    PROC  WELD_A_SQUARE_ANCHOR()
        !!!NOW HAS THE WOBJ WRINKLE REMOVED 02-05-18!!!!!!!
        !!!!!THIS PROGRAM IS now revised Square_Anchor TO GET SEARCHED IN POSITION 02-05-18!!!!!!!
        !!!!! nozzle search version 02-05-18!!!!!!!!!!!
        !!!!!!!!!!!!!!!!REVISED 03-16-18 to add anchor_back X searches!!!!!
        ActUnit STN1;
		AccSet 40, 40;
        MoveJ pjthomeSTA1zero, vCellSpeed, fine, tWeldGun\WObj:=wobj0;
        MoveJ Offs(SP_AGBY_S,0,-300,50), v400, z5, tWeldGun\WObj:=wobjHanchor_BACK;
		MoveL Offs(SP_AGBY_S,0,-100,50), v300, z5, tWeldGun\WObj:=wobjHanchor_BACK;
        MoveL SP_AGBY_S, v200, z5, tWeldGun\WObj:=wobjHanchor_BACK;
		Search_1D SR_AGB_Y\SearchStop:=AG_BY, SP_AGBY_S, SP_AGBY_E, v50, tWeldGun\WObj:=wobjHanchor_BACK\SchSpeed:=10;
  		MoveL AG_BY, v50, fine, tWeldGun\WObj:=wobjHanchor_BACK;
  		WaitTime\InPos, 1;
  		AG_BY_DEFLECTION := CRobT(\Tool:=tWeldGun\WObj:=obSTN1);
  		WaitTime\InPos, 1;
		AG_BY_DEFLECTION.trans.y := AG_BY_DEFLECTION.trans.y + NOZZLE_RADIUS;
        WaitTime\InPos, 0.2;
        TPWrite "SR_AGB_Y DEFLECTION:="\Pos:=SR_AGB_Y.trans;
		MoveL SP_AGBY_S, v300, z5, tWeldGun\WObj:=wobjHanchor_BACK;
        MoveL SP_AHBY_S, v300, z5, tWeldGun\WObj:=wobjHanchor_BACK;
		Search_1D SR_AHB_Y\SearchStop:=AH_BY, SP_AHBY_S, SP_AHBY_E, v50, tWeldGun\WObj:=wobjHanchor_BACK\SchSpeed:=10;
  		MoveL AH_BY, v50, fine, tWeldGun\WObj:=wobjHanchor_BACK;
  		WaitTime\InPos, 1;
		AH_BY_DEFLECTION := CRobT(\Tool:=tWeldGun\WObj:=obSTN1);
  		WaitTime\InPos, 1;
		AH_BY_DEFLECTION.trans.y := AH_BY_DEFLECTION.trans.y + NOZZLE_RADIUS;
        WaitTime\InPos, 0.2;
		TPWrite "SR_AHB_Y DEFLECTION:="\Pos:=SR_AHB_Y.trans;
		MoveL SP_AHBY_S, v200, z5, tWeldGun\WObj:=wobjHanchor_BACK;
	    MoveJ Offs(SP_AHBY_S,0,-275,75), v500, z5, tWeldGun\WObj:=wobjHanchor_BACK;
	    MoveJ Offs(SP_AHBY_S,0,-425,125), v500, z5, tWeldGun\WObj:=wobjHanchor_BACK;
	    MoveJ Offs(SP_AHBY_S,0,-625,125), v500, z5, tWeldGun\WObj:=wobjHanchor_BACK;
		MoveJ Offs(SP_GX_S,0,-400,50), v500, z5, tWeldGun\WObj:=wobjHanchor_BACK;
		MoveJ Offs(SP_GX_S,0,-200,50), v500, z5, tWeldGun\WObj:=wobjHanchor_BACK;
		MoveL Offs(SP_GX_S,0,-200,50), v500, z5, tWeldGun\WObj:=wobjHanchor_BACK;
		MoveL Offs(SP_GX_S,0,-50,50), v500, z5, tWeldGun\WObj:=wobjHanchor_BACK;
        MoveL SP_GX_S, v200, z1, tWeldGun\WObj:=wobjHanchor;
		Search_1D SR_AG_X\SearchStop:=AG_X, SP_GX_S, SP_GX_E, v50, tWeldGun\WObj:=wobjHanchor\SchSpeed:=10;
        TPWrite "SR_AG_X :="\Pos:=SR_AG_X.trans;
		MoveL SP_GX_S, v200, z1, tWeldGun\WObj:=wobjHanchor;
        MoveL SP_AGBZ_S, v200, z1, tWeldGun\WObj:=wobjHanchor_BACK;
	    Search_1D SR_AGB_Z\SearchStop:=AG_BZ, SP_AGBZ_S, SP_AGBZ_E, v50, tWeldGun\WObj:=wobjHanchor_BACK\SchSpeed:=10;
     	MoveL AG_BZ, v50, fine, tWeldGun\WObj:=wobjHanchor_BACK;
  		WaitTime\InPos, 1;
		AG_BZ_DEFLECTION := CRobT(\Tool:=tWeldGun\WObj:=obSTN1);
        WaitTime\InPos, .1;
        TPWrite "SR_AGB_Z DEFLECTION:="\Pos:=SR_AGB_Z.trans;
        MoveL SP_AGBZ_S, v200, z1, tWeldGun\WObj:=wobjHanchor_BACK;
        MoveL Offs(SP_AGBZ_S,0,-325,50), v200, z1, tWeldGun\WObj:=wobjHanchor_BACK;
        MoveJ Offs(SP_AHBZ_S,0,-325,50), v200, z1, tWeldGun\WObj:=wobjHanchor_BACK;
        MoveL SP_AHBZ_S, v200, z1, tWeldGun\WObj:=wobjHanchor_BACK;
	    Search_1D SR_AHB_Z\SearchStop:=AH_BZ, SP_AHBZ_S, SP_AHBZ_E, v50, tWeldGun\WObj:=wobjHanchor_BACK\SchSpeed:=10;
     	MoveL AH_BZ, v50, fine, tWeldGun\WObj:=wobjHanchor_BACK;
  		WaitTime\InPos, 1;
		AH_BZ_DEFLECTION := CRobT(\Tool:=tWeldGun\WObj:=obSTN1);
        WaitTime\InPos, .1;
        TPWrite "SR_AHB_Z DEFLECTION:="\Pos:=SR_AHB_Z.trans;
        MoveL SP_AHBZ_S, v200, z1, tWeldGun\WObj:=wobjHanchor_BACK;
        MoveL SP_HX_S, v200, z1, tWeldGun\WObj:=wobjHanchor;
		Search_1D SR_AH_X\SearchStop:=AH_X, SP_HX_S, SP_HX_E, v50, tWeldGun\WObj:=wobjHanchor\SchSpeed:=10;
        TPWrite "SR_AH_X :="\Pos:=SR_AH_X.trans;
		MoveL SP_HX_S, v200, z1, tWeldGun\WObj:=wobjHanchor;
		MoveL Offs(SP_AHBZ_S,0,-125,50), v200, z5, tWeldGun\WObj:=wobjHanchor_BACK;
		MoveL Offs(SP_AHBZ_S,0,-500,100), v200, z5, tWeldGun\WObj:=wobjHanchor_BACK;
        RESET_ANCHOR_BACK_WOBJ;
        SET_ANCHOR_X AH_X ;
        SET_ANCHOR_X AG_X ;
        TPWrite "NOW WORKING ON WELD 'AH_BACK'";
		MoveJ Offs(AH201,-150,-250,-10), vExtMax, z1, tWeldGun\WObj:=wobjHanchor_BACK_H;
		MoveL RelTool(AH200,0,0,-20), v200, z1, tWeldGun\WObj:=wobjHanchor_BACK_H;
		ArcLStart AH200, v100, smHCYLANCH, wdHCYLANCH\Weave:=wvHCYLANCH, fine, tWeldGun\WObj:=wobjHanchor_BACK_H\Track:=trHCYLANCHhiteonly;
		ArcL AH201, v100, smHCYLANCH, wdHCYLANCH\Weave:=wvHCYLANCH, z10, tWeldGun\WObj:=wobjHanchor_BACK_H\Track:=trHCYLANCHhiteonly;
		ArcLEnd AH202, v100, smHCYLANCH, wdHCYLANCH\Weave:=wvHCYLANCH, z10, tWeldGun\WObj:=wobjHanchor_BACK_H\Track:=trHCYLANCHhiteonly;
		MoveL RelTool(AH202,0,0,-100), v200, z1, tWeldGun\WObj:=wobjHanchor_BACK;
		MoveJ Offs(AH202,-50,-150,0), vExtMax, z1, tWeldGun\WObj:=wobjHanchor_BACK;
	    TPWrite "NOW WORKING ON WELD 'AG_BACK'";
		MoveL Offs(AG201,50,-150,0), vExtMax, z1, tWeldGun\WObj:=wobjHanchor_BACK;
		MoveL RelTool(AG200,0,0,-20), v200, z1, tWeldGun\WObj:=wobjHanchor_BACK;
		ArcLStart AG200, v100, smHCYLANCH, wdHCYLANCH\Weave:=wvHCYLANCH, fine, tWeldGun\WObj:=wobjHanchor_BACK_G\Track:=trHCYLANCHhiteonly;
		ArcL AG201, v100, smHCYLANCH, wdHCYLANCH\Weave:=wvHCYLANCH, z10, tWeldGun\WObj:=wobjHanchor_BACK_G\Track:=trHCYLANCHhiteonly;
		ArcLEnd AG202, v100, smHCYLANCH, wdHCYLANCH\Weave:=wvHCYLANCH, z10, tWeldGun\WObj:=wobjHanchor_BACK_G\Track:=trHCYLANCHhiteonly;
		MoveL RelTool(AG202,0,0,-100), v200, z1, tWeldGun\WObj:=wobjHanchor_BACK;
		MoveL pairanchor11, v500, z1, tWeldGun\WObj:=wobjHanchor_BACK;
		MoveJ pjthomeSTA1zero, vCellSpeed, fine, tWeldGun\WObj:=wobj0;
		!MoveL Offs(AG202,300,-650,50), v200, z1, tWeldGun\WObj:=wobjHanchor_BACK;
		!CutWire;
		ActUnit STN1;
        MoveJ Offs(SP_AGFY_S,0,800,200), v1000, z5, tWeldGun\WObj:=wobjHanchor_FRONT;
        MoveJ Offs(SP_AGFY_S,0,150,100), v400, z5, tWeldGun\WObj:=wobjHanchor_FRONT;
        MoveL SP_AGFY_S, v200, z1, tWeldGun\WObj:=wobjHanchor_FRONT;
		Search_1D SR_AGF_Y1\SearchStop:=AG_FY, SP_AGFY_S, SP_AGFY_E, v50, tWeldGun\WObj:=wobjHanchor_FRONT\SchSpeed:=10;
        TPWrite "SR_AGF_Y1 DEFLECTION:="\Pos:=SR_AGF_Y1.trans;
		Search_1D SR_AGF_Y2\SearchStop:=AG_FY, SP_AGFY_S, SP_AGFY_E, v50, tWeldGun\WObj:=wobjHanchor_FRONT\SchSpeed:=10;
        TPWrite "SR_AGF_Y2 DEFLECTION:="\Pos:=SR_AGF_Y2.trans;
        MoveL AG_FY, v50, fine, tWeldGun\WObj:=wobjHanchor_FRONT;
  		WaitTime\InPos, 1;
		AG_FY_DEFLECTION := CRobT(\Tool:=tWeldGun\WObj:=obSTN1);
        WaitTime\InPos, 1;
        AG_FY_DEFLECTION.trans.y := AG_FY_DEFLECTION.trans.y - NOZZLE_RADIUS;
        WaitTime\InPos, 0.2;
		MoveL SP_AGFY_S, v300, z1, tWeldGun\WObj:=wobjHanchor_FRONT;
        MoveL SP_AHFY_S, v300, z1, tWeldGun\WObj:=wobjHanchor_FRONT;
		Search_1D SR_AHF_Y1\SearchStop:=AH_FY, SP_AHFY_S, SP_AHFY_E, v50, tWeldGun\WObj:=wobjHanchor_FRONT\SchSpeed:=10;
        TPWrite "SR_AHF_Y1 DEFLECTION:="\Pos:=SR_AHF_Y1.trans;
		Search_1D SR_AHF_Y2\SearchStop:=AH_FY, SP_AHFY_S, SP_AHFY_E, v50, tWeldGun\WObj:=wobjHanchor_FRONT\SchSpeed:=10;
  		TPWrite "SR_AHF_Y2 DEFLECTION:="\Pos:=SR_AHF_Y2.trans;
        MoveL AH_FY, v50, fine, tWeldGun\WObj:=wobjHanchor_FRONT;
  		WaitTime\InPos, 1;
		AH_FY_DEFLECTION := CRobT(\Tool:=tWeldGun\WObj:=obSTN1);
        WaitTime\InPos, 1;
        AH_FY_DEFLECTION.trans.y := AH_FY_DEFLECTION.trans.y - NOZZLE_RADIUS;
        WaitTime\InPos, 0.2;
	    ! POSSIBLY NEED TO ADD A "Y" DISPLACEMENT TO KEEP THE "Z" SEARCH ON THE NOZZLE
        SR_AHF_Y2.TRANS.Y := SR_AHF_Y1.TRANS.Y;
		PDispSet SR_AHF_Y2;
		MoveL Offs(SP_AHFY_S,0,50,0), v300, z1, tWeldGun\WObj:=wobjHanchor_FRONT;
		MoveL Offs(SP_AHFY_S,0,250,100), v300, z1, tWeldGun\WObj:=wobjHanchor_FRONT;
        MoveJ Offs(SP_AHFZ_S,0,400,50), v300, z1, tWeldGun\WObj:=wobjHanchor_FRONT;
        MoveJ Offs(SP_AHFZ_S,0,100,50), v300, z1, tWeldGun\WObj:=wobjHanchor_FRONT;
		MoveL SP_AHFZ_S, v200, z1, tWeldGun\WObj:=wobjHanchor_FRONT;
        Search_1D SR_AHF_Z\SearchStop:=AH_FZ, SP_AHFZ_S, SP_AHFZ_E, v50, tWeldGun\WObj:=wobjHanchor_FRONT\SchSpeed:=10;
  		MoveL AH_FZ, v50, fine, tWeldGun\WObj:=wobjHanchor_FRONT;
        WaitTime\InPos, 1;
        AH_FZ_DEFLECTION := CRobT(\Tool:=tWeldGun\WObj:=obSTN1);
        WaitTime\InPos, 1;
        TPWrite "SR_AGF_Z DEFLECTION:="\Pos:=SR_AGF_Z.trans;
		MoveL SP_AHFZ_S, v200, z1, tWeldGun\WObj:=wobjHanchor_FRONT;
        ! ADDED X SEARCH HERE
		MoveJ SP_AHFX_S, v200, z1, tWeldGun\WObj:=wobjHanchor_FRONT;
        Search_1D SR_AHF_X\SearchStop:=AH_X, SP_AHFX_S, SP_AHFX_E, v50, tWeldGun\WObj:=wobjHanchor_FRONT\SchSpeed:=10;
		MoveL SP_AHFZ_S, v200, z1, tWeldGun\WObj:=wobjHanchor_FRONT;
        ! POSSIBLY NEED TO ADD A "Y" DISPLACEMENT TO KEEP THE "Z" SEARCH ON THE NOZZLE
        SR_AGF_Y2.TRANS.Y := SR_AGF_Y1.TRANS.Y;
		PDispSet SR_AGF_Y2;
        MoveJ SP_AGFZ_S, v200, z1, tWeldGun\WObj:=wobjHanchor_FRONT;
		Search_1D SR_AGF_Z\SearchStop:=AG_FZ, SP_AGFZ_S, SP_AGFZ_E, v50, tWeldGun\WObj:=wobjHanchor_FRONT\SchSpeed:=10;
   		MoveL AG_FZ, v50, fine, tWeldGun\WObj:=wobjHanchor_FRONT;
        WaitTime\InPos, 1;
        AG_FZ_DEFLECTION := CRobT(\Tool:=tWeldGun\WObj:=obSTN1);
        WaitTime\InPos, 1;
        TPWrite "SR_AGF_Z DEFLECTION:="\Pos:=SR_AGF_Z.trans;
		MoveL SP_AGFZ_S, v200, z1, tWeldGun\WObj:=wobjHanchor_FRONT;
        ! ADDED X SEARCH HERE
 		MoveL SP_AGFX_S, v200, z1, tWeldGun\WObj:=wobjHanchor_FRONT;
        Search_1D SR_AGF_X\SearchStop:=AG_X, SP_AGFX_S, SP_AGFX_E, v50, tWeldGun\WObj:=wobjHanchor_FRONT\SchSpeed:=10;
		MoveL SP_AGFZ_S, v200, z1, tWeldGun\WObj:=wobjHanchor_FRONT;
        MoveL OFFS(SP_AGFZ_S,0,100,75), v200, z1, tWeldGun\WObj:=wobjHanchor_FRONT;
        MoveL OFFS(SP_AGFZ_S,0,600,75), v400, z1, tWeldGun\WObj:=wobjHanchor_FRONT;
        FRONT_ANCHOR_ROTATION_DEFLECTION  wobjHanchor_FRONT_H, AH_FY_DEFLECTION, AH_FY, AH_FZ_DEFLECTION, AH_FZ;
        FRONT_ANCHOR_ROTATION_DEFLECTION  wobjHanchor_FRONT_G, AG_FY_DEFLECTION, AG_FY, AG_FZ_DEFLECTION, AG_FZ;
        FRONT_ANCHOR_TRANS_DEFLECTION wobjHanchor_FRONT_G, AG_FY_DEFLECTION, AG_FZ_DEFLECTION, AG_FY, AG_FZ  ;
        FRONT_ANCHOR_TRANS_DEFLECTION wobjHanchor_FRONT_H, AH_FY_DEFLECTION, AH_FZ_DEFLECTION, AH_FY, AH_FZ  ;
        SET_ANCHOR_X AG_X;
        SET_ANCHOR_X AH_X;
        MoveJ Offs(AG206,150,300,50), v400, z1, tWeldGun\WObj:=wobjHanchor_FRONT_G;
		MoveL RelTool(AG206,0,0,-30), v200, z1, tWeldGun\WObj:=wobjHanchor_FRONT_G;
        ArcLStart AG206, v100, smHCYLANCH, wdHCYLANCH\Weave:=wvHCYLANCH, fine, tWeldGun\WObj:=wobjHanchor_FRONT_G\Track:=trHCYLANCHhiteonly;
		ArcL AG207, v100, smHCYLANCH, wdHCYLANCH\Weave:=wvHCYLANCH, z10, tWeldGun\WObj:=wobjHanchor_FRONT_G\Track:=trHCYLANCHhiteonly;
		ArcLEnd AG208, v100, smHCYLANCH, wdHCYLANCH\Weave:=wvHCYLANCH, z10, tWeldGun\WObj:=wobjHanchor_FRONT_G\Track:=trHCYLANCHhiteonly;
		MoveL RelTool(AG208,0,0,-10), v200, z1, tWeldGun\WObj:=wobjHanchor_FRONT_G;
		MoveL RelTool(AG206,0,0,-150), vExtMax, z1, tWeldGun\WObj:=wobjHanchor_FRONT_G;
		MoveL Offs(AG206,150,250,50), vExtMax, z1, tWeldGun\WObj:=wobjHanchor_FRONT_G;
		MoveJ Offs(AG220,150,350,50), vExtMax, z1, tWeldGun\WObj:=wobjHanchor_FRONT_G;
		MoveJ Offs(AG220,50,350,50), vExtMax, z1, tWeldGun\WObj:=wobjHanchor_FRONT_G;
   		MoveJ Offs(AG220,50,50,50), vExtMax, z1, tWeldGun\WObj:=wobjHanchor_FRONT_G;
    	MoveL RelTool(AG220,0,0,-15), vExtMax, fine, tWeldGun\WObj:=wobjHanchor_FRONT_G;
		ArcLStart AG220, v100, smHCYLANCH, wdHCYLANCH\Weave:=wv0, fine, tWeldGun\WObj:=wobjHanchor_FRONT_G\Track:=trHCYLANCHhiteonly;
		ArcL AG219, v100, smHCYLANCH, wdHCYLANCH\Weave:=wv0, z10, tWeldGun\WObj:=wobjHanchor_FRONT_G\Track:=trHCYLANCHhiteonly;
		ArcLEnd AG218, v100, smHCYLANCH, wdHCYLANCH\Weave:=wv0, z10, tWeldGun\WObj:=wobjHanchor_FRONT_G\Track:=trHCYLANCHhiteonly;
		MoveL RelTool(AG218,0,-5,-15), vExtMax, fine, tWeldGun\WObj:=wobjHanchor_FRONT_G;
		MoveL RelTool(AG219,0,-5,-15), vExtMax, fine, tWeldGun\WObj:=wobjHanchor_FRONT_G;
		MoveL RelTool(AG220,0,-10,-15), vExtMax, fine, tWeldGun\WObj:=wobjHanchor_FRONT_G;
  		MoveJ Offs(AG220,50,75,50), vExtMax, z1, tWeldGun\WObj:=wobjHanchor_FRONT_G;
  		MoveJ Offs(AG220,150,350,50), vExtMax, z1, tWeldGun\WObj:=wobjHanchor_FRONT_G;
  		IF bAnchor_Lite = TRUE THEN
  			GOTO Short_Cut;
  		ENDIF
        MoveJ Offs(AG203,75,350,-25), vExtMax, z1, tWeldGun\WObj:=wobjHanchor_FRONT_G;
		MoveL Offs(AG203,25,25,-25), vExtMax, z1, tWeldGun\WObj:=wobjHanchor_FRONT_G;
		MoveL RelTool(AG203,0,0,-15), vExtMax, fine, tWeldGun\WObj:=wobjHanchor_FRONT_G;
		ArcLStart AG203, v100, smHCYLANCH, wdHCYLANCH\Weave:=wvHCYLANCH, z0, tWeldGun\WObj:=wobjHanchor_FRONT_G\Track:=trHCYLANCHhiteonly;
		ArcL AG204, v100, smHCYLANCH, wdHCYLANCH\Weave:=wvHCYLANCH, z10, tWeldGun\WObj:=wobjHanchor_FRONT_G\Track:=trHCYLANCHhiteonly;
		ArcLEnd AG205, v100, smHCYLANCH, wdHCYLANCH\Weave:=wvHCYLANCH, fine, tWeldGun\WObj:=wobjHanchor_FRONT_G\Track:=trHCYLANCHhiteonly;
		MoveL RelTool(AG204,10,0,-15), vExtMax, fine, tWeldGun\WObj:=wobjHanchor_FRONT_G;
		MoveL Offs(AG204,30,100,-25), vExtMax, fine, tWeldGun\WObj:=wobjHanchor_FRONT_G;
		MoveL Offs(AG204,75,200,-40), vExtMax, fine, tWeldGun\WObj:=wobjHanchor_FRONT_G;
		Short_Cut:
		MoveL Offs(AG205,850,450,100), vExtMax, fine, tWeldGun\WObj:=wobjHanchor_FRONT_G;
 		MoveJ Offs(AH206,-150,250,100), vExtMax, z1, tWeldGun\WObj:=wobjHanchor_FRONT_H;
 		MoveL RelTool(AH206,0,0,-20), v200, z1, tWeldGun\WObj:=wobjHanchor_FRONT_H;
        ArcLStart AH206, v100, smHCYLANCH, wdHCYLANCH\Weave:=wvHCYLANCH, z0, tWeldGun\WObj:=wobjHanchor_FRONT_H\Track:=trHCYLANCHhiteonly;
		ArcL AH207, v100, smHCYLANCH, wdHCYLANCH\Weave:=wvHCYLANCH, z10, tWeldGun\WObj:=wobjHanchor_FRONT_H\Track:=trHCYLANCHhiteonly;
		ArcLEnd AH208, v100, smHCYLANCH, wdHCYLANCH\Weave:=wvHCYLANCH, fine, tWeldGun\WObj:=wobjHanchor_FRONT_H\Track:=trHCYLANCHhiteonly;
		MoveL RelTool(AH208,0,0,-10), v200, z1, tWeldGun\WObj:=wobjHanchor_FRONT_H;
		MoveL RelTool(AH206,0,0,-150), vExtMax, z1, tWeldGun\WObj:=wobjHanchor_FRONT_H;
		MoveJ Offs(AH206,-150,250,50), vExtMax, z1, tWeldGun\WObj:=wobjHanchor_FRONT_H;
		MoveJ Offs(AH220,-150,250,50), vExtMax, z1, tWeldGun\WObj:=wobjHanchor_FRONT_H;
		MoveL RelTool(AH220,-3,3,-15), vExtMax, fine, tWeldGun\WObj:=wobjHanchor_FRONT_H;
  		ArcLStart AH220, v100, smHCYLANCH, wdHCYLANCH\Weave:=wv0, fine, tWeldGun\WObj:=wobjHanchor_FRONT_H\Track:=trHCYLANCHhiteonly;
		ArcL AH219, v100, smHCYLANCH, wdHCYLANCH\Weave:=wv0, z10, tWeldGun\WObj:=wobjHanchor_FRONT_H\Track:=trHCYLANCHhiteonly;
		ArcLEnd AH218, v100, smHCYLANCH, wdHCYLANCH\Weave:=wv0, z10, tWeldGun\WObj:=wobjHanchor_FRONT_H\Track:=trHCYLANCHhiteonly;
		PDispOff;
		MoveL RelTool(AH218,-0,3,-15), v200, fine, tWeldGun\WObj:=wobjHanchor_FRONT_H;
		MoveL RelTool(AH219,-0,3,-15), v200, fine, tWeldGun\WObj:=wobjHanchor_FRONT_H;
		MoveL RelTool(AH220,-8,0,-15), v200, fine, tWeldGun\WObj:=wobjHanchor_FRONT_H;
  		MoveJ Offs(AH220,-100,250,0), vExtMax, z1, tWeldGun\WObj:=wobjHanchor_FRONT_H;
  		MoveJ Offs(AH206,-100,250,0), vExtMax, z1, tWeldGun\WObj:=wobjHanchor_FRONT_H;
  		IF bAnchor_Lite = TRUE THEN
  			GOTO Shorter_Cut;
  		ENDIF
       	MoveL Offs(AH203,-50,350,-50), vExtMax, z1, tWeldGun\WObj:=wobjHanchor_FRONT_H;
		MoveL Offs(AH203,-25,25,-25), vExtMax, z1, tWeldGun\WObj:=wobjHanchor_FRONT_H;
		MoveL RelTool(AH203,8,0,-15), v200, z1, tWeldGun\WObj:=wobjHanchor_FRONT_H;
		ArcLStart AH203, v100, smHCYLANCH, wdHCYLANCH\Weave:=wvHCYLANCH, fine, tWeldGun\WObj:=wobjHanchor_FRONT_H\Track:=trHCYLANCHhiteonly;
		ArcL AH204, v100, smHCYLANCH, wdHCYLANCH\Weave:=wvHCYLANCH, z10, tWeldGun\WObj:=wobjHanchor_FRONT_H\Track:=trHCYLANCHhiteonly;
		ArcLEnd AH205, v100, smHCYLANCH, wdHCYLANCH\Weave:=wvHCYLANCH, fine, tWeldGun\WObj:=wobjHanchor_FRONT_H\Track:=trHCYLANCHhiteonly;
		MoveL RelTool(AH204,8,0,-15), v200, z1, tWeldGun\WObj:=wobjHanchor_FRONT_H;
		MoveL RelTool(AH203,8,0,-15), v200, z1, tWeldGun\WObj:=wobjHanchor_FRONT_H;
		MoveL Offs(AH203,-50,50,-25), vExtMax, z1, tWeldGun\WObj:=wobjHanchor_FRONT_H;
		MoveL Offs(AH203,-100,150,-25), vExtMax, z1, tWeldGun\WObj:=wobjHanchor_FRONT_H;
		MoveL Offs(AH203,-250,250,-25), vExtMax, fine, tWeldGun\WObj:=wobjHanchor_FRONT_H;
		Shorter_Cut:
        MoveL Offs(AH208,-350,550,20), vExtMax, z1, tWeldGun\WObj:=wobjHanchor_FRONT_H;
        MoveJ pjthomeSTA1zero, vCellSpeed, fine, tWeldGun\WObj:=wobj0;
        LABEL:
    ENDPROC

    PROC  WELD_A_TAPERED_SQUARE_ANCHOR()
        !THE WOBJ WRINKLE HAS BEEN REMOVED FROM THIS PROC 12-01-17!!!!!!!!!!!
        !!!!!THIS PROGRAM IS now revised Tapered_Square_Anchor TO GET SEARCHED IN POSITION 12-01-17!!!!!!!
        !!!!! nozzle search version 12-01-17!!!!!!!!!!!
        !!!!!!!!!!!!!!!!REVISED 03-16-18 to add anchor_back X searches!!!!!
        ActUnit STN1;
		AccSet 40, 40;
        MoveJ pjthomeSTA1zero, vCellSpeed, fine, tWeldGun\WObj:=wobj0;
        MoveJ Offs(SP_AGBY_S,0,-300,50), v500, z5, tWeldGun\WObj:=wobjHanchor_BACK;
		MoveL Offs(SP_AGBY_S,0,-100,50), v500, z5, tWeldGun\WObj:=wobjHanchor_BACK;
        MoveL SP_AGBY_S, v500, z5, tWeldGun\WObj:=wobjHanchor_BACK;
		Search_1D SR_AGB_Y\SearchStop:=AG_BY, SP_AGBY_S, SP_AGBY_E, v50, tWeldGun\WObj:=wobjHanchor_BACK\SchSpeed:=10;
  		MoveL AG_BY, v50, fine, tWeldGun\WObj:=wobjHanchor_BACK;
  		WaitTime\InPos, 1;
		AG_BY_DEFLECTION := CRobT(\Tool:=tWeldGun\WObj:=obSTN1);
        WaitTime\InPos, 1;
        AG_BY_DEFLECTION.trans.y := AG_BY_DEFLECTION.trans.y + NOZZLE_RADIUS;
        WaitTime\InPos, 0.2;
        TPWrite "SR_AGB_Y DEFLECTION:="\Pos:=SR_AGB_Y.trans;
		MoveL SP_AGBY_S, v500, z5, tWeldGun\WObj:=wobjHanchor_BACK;
        MoveL SP_AHBY_S, v500, z5, tWeldGun\WObj:=wobjHanchor_BACK;
		Search_1D SR_AHB_Y\SearchStop:=AH_BY, SP_AHBY_S, SP_AHBY_E, v50, tWeldGun\WObj:=wobjHanchor_BACK\SchSpeed:=10;
  		MoveL AH_BY, v50, fine, tWeldGun\WObj:=wobjHanchor_BACK;
  		WaitTime\InPos, 1;
		AH_BY_DEFLECTION := CRobT(\Tool:=tWeldGun\WObj:=obSTN1);
        WaitTime\InPos, 1;
        AH_BY_DEFLECTION.trans.y := AH_BY_DEFLECTION.trans.y + NOZZLE_RADIUS;
        WaitTime\InPos, 0.2;
		TPWrite "SR_AHB_Y DEFLECTION:="\Pos:=SR_AHB_Y.trans;
		MoveL SP_AHBY_S, v500, z5, tWeldGun\WObj:=wobjHanchor_BACK;
	    MoveJ Offs(SP_AHBY_S,0,-275,75), v500, z5, tWeldGun\WObj:=wobjHanchor_BACK;
	    MoveJ Offs(SP_AHBY_S,0,-575,175), v500, z5, tWeldGun\WObj:=wobjHanchor_BACK;
	    MoveJ Offs(SP_GX_S,0,-400,150), v500, z5, tWeldGun\WObj:=wobjHanchor_BACK;
		MoveJ Offs(SP_GX_S,0,-300,50), v500, z5, tWeldGun\WObj:=wobjHanchor_BACK;
		MoveL Offs(SP_GX_S,0,-200,50), v500, z5, tWeldGun\WObj:=wobjHanchor_BACK;
		MoveL Offs(SP_GX_S,0,-50,50), v500, z5, tWeldGun\WObj:=wobjHanchor_BACK;
        MoveL SP_GX_S, v500, z1, tWeldGun\WObj:=wobjHanchor;
		Search_1D SR_AG_X\SearchStop:=AG_X, SP_GX_S, SP_GX_E, v50, tWeldGun\WObj:=wobjHanchor\SchSpeed:=10;
        TPWrite "SR_AG_X :="\Pos:=SR_AG_X.trans;
		MoveL SP_GX_S, v500, z1, tWeldGun\WObj:=wobjHanchor;
        MoveL SP_AGBZ_S, v500, z1, tWeldGun\WObj:=wobjHanchor_BACK;
	    Search_1D SR_AGB_Z\SearchStop:=AG_BZ, SP_AGBZ_S, SP_AGBZ_E, v50, tWeldGun\WObj:=wobjHanchor_BACK\SchSpeed:=10;
     	MoveL AG_BZ, v50, fine, tWeldGun\WObj:=wobjHanchor_BACK;
  		WaitTime\InPos, 1;
		AG_BZ_DEFLECTION := CRobT(\Tool:=tWeldGun\WObj:=obSTN1);
        WaitTime\InPos, 1;
        TPWrite "SR_AGB_Z DEFLECTION:="\Pos:=SR_AGB_Z.trans;
        MoveL SP_AGBZ_S, v500, z1, tWeldGun\WObj:=wobjHanchor_BACK;
        MoveL Offs(SP_AGBZ_S,100,-325,50), v500, z1, tWeldGun\WObj:=wobjHanchor_BACK;
        MoveJ Offs(SP_AHBZ_S,0,-325,50), v500, z1, tWeldGun\WObj:=wobjHanchor_BACK;
        MoveL SP_AHBZ_S, v500, z1, tWeldGun\WObj:=wobjHanchor_BACK;
	    Search_1D SR_AHB_Z\SearchStop:=AH_BZ, SP_AHBZ_S, SP_AHBZ_E, v50, tWeldGun\WObj:=wobjHanchor_BACK\SchSpeed:=10;
     	MoveL AH_BZ, v50, fine, tWeldGun\WObj:=wobjHanchor_BACK;
  		WaitTime\InPos, 1;
		AH_BZ_DEFLECTION := CRobT(\Tool:=tWeldGun\WObj:=obSTN1);
        WaitTime\InPos, 1;
        TPWrite "SR_AHB_Z DEFLECTION:="\Pos:=SR_AHB_Z.trans;
        MoveL SP_AHBZ_S, v500, z1, tWeldGun\WObj:=wobjHanchor_BACK;
        MoveL SP_HX_S, v500, z1, tWeldGun\WObj:=wobjHanchor;
		Search_1D SR_AH_X\SearchStop:=AH_X, SP_HX_S, SP_HX_E, v50, tWeldGun\WObj:=wobjHanchor\SchSpeed:=10;
        TPWrite "SR_AH_X :="\Pos:=SR_AH_X.trans;
		MoveL SP_HX_S, v500, z1, tWeldGun\WObj:=wobjHanchor;
		MoveL Offs(SP_AHBZ_S,0,-125,50), v500, z5, tWeldGun\WObj:=wobjHanchor_BACK;
		MoveL Offs(SP_AHBZ_S,0,-500,100), v500, z5, tWeldGun\WObj:=wobjHanchor_BACK;
	    RESET_ANCHOR_BACK_WOBJ;
        SET_ANCHOR_X AG_X;
        SET_ANCHOR_X AH_X;
        TPWrite "NOW WORKING ON WELD 'AH_BACK'";
		MoveJ Offs(AH401,-150,-250,-10), vExtMax, z1, tWeldGun\WObj:=wobjHanchor_BACK_H;
		MoveL RelTool(AH400,0,0,-20), v500, z1, tWeldGun\WObj:=wobjHanchor_BACK_H;
		ArcLStart AH400, v100, smHCYLANCH, wdHCYLANCH\Weave:=wvHCYLANCH, fine, tWeldGun\WObj:=wobjHanchor_BACK_H\Track:=trHCYLANCHhiteonly;
		ArcL AH401, v100, smHCYLANCH, wdHCYLANCH\Weave:=wvHCYLANCH, z10, tWeldGun\WObj:=wobjHanchor_BACK_H\Track:=trHCYLANCHhiteonly;
		ArcLEnd AH402, v100, smHCYLANCH, wdHCYLANCH\Weave:=wvHCYLANCH, z10, tWeldGun\WObj:=wobjHanchor_BACK_H\Track:=trHCYLANCHhiteonly;
		MoveL RelTool(AH402,0,0,-100), v200, z1, tWeldGun\WObj:=wobjHanchor_BACK;
		MoveJ Offs(AH402,-50,-150,0), vExtMax, z1, tWeldGun\WObj:=wobjHanchor_BACK;
	    TPWrite "NOW WORKING ON WELD 'AG_BACK'";
		MoveL Offs(AG401,50,-150,0), vExtMax, z1, tWeldGun\WObj:=wobjHanchor_BACK;
		MoveL RelTool(AG400,0,0,-20), v500, z1, tWeldGun\WObj:=wobjHanchor_BACK;
		ArcLStart AG400, v100, smHCYLANCH, wdHCYLANCH\Weave:=wvHCYLANCH, fine, tWeldGun\WObj:=wobjHanchor_BACK_G\Track:=trHCYLANCHhiteonly;
		ArcL AG401, v100, smHCYLANCH, wdHCYLANCH\Weave:=wvHCYLANCH, z10, tWeldGun\WObj:=wobjHanchor_BACK_G\Track:=trHCYLANCHhiteonly;
		ArcLEnd AG402, v100, smHCYLANCH, wdHCYLANCH\Weave:=wvHCYLANCH, z10, tWeldGun\WObj:=wobjHanchor_BACK_G\Track:=trHCYLANCHhiteonly;
		MoveL RelTool(AG402,0,0,-100), v500, z1, tWeldGun\WObj:=wobjHanchor_BACK;
		MoveL RelTool(AG402,0,0,-300), v500, z1, tWeldGun\WObj:=wobjHanchor_BACK;
		!MoveL Offs(AG402,300,-650,50), v200, z1, tWeldGun\WObj:=wobjHanchor_BACK;
		MoveJ pjthomeSTA1zero, vCellSpeed, fine, tWeldGun\WObj:=wobj0;
		!CutWire;
		ActUnit STN1;
        !!!!!!!!!!!  WILLIE MAKE IT   !!!!!!!!!!!
        MoveJ Offs(SP_AGFY_S,0,800,0), v1000, z5, tWeldGun\WObj:=wobjHanchor_FRONT;
        !!!!!!!!!!!  WILLIE MAKE IT   !!!!!!!!!!!
        MoveJ Offs(SP_AGFY_S,0,150,0), v500, z5, tWeldGun\WObj:=wobjHanchor_FRONT;
        MoveL SP_AGFY_S, v500, z1, tWeldGun\WObj:=wobjHanchor_FRONT;
		Search_1D SR_AGF_Y1\SearchStop:=AG_FY, SP_AGFY_S, SP_AGFY_E, v50, tWeldGun\WObj:=wobjHanchor_FRONT\SchSpeed:=10;
        TPWrite "SR_AGF_Y1 DEFLECTION:="\Pos:=SR_AGF_Y1.trans;
		Search_1D SR_AGF_Y2\SearchStop:=AG_FY, SP_AGFY_S, SP_AGFY_E, v50, tWeldGun\WObj:=wobjHanchor_FRONT\SchSpeed:=10;
        TPWrite "SR_AGF_Y2 DEFLECTION:="\Pos:=SR_AGF_Y2.trans;
        MoveL AG_FY, v50, fine, tWeldGun\WObj:=wobjHanchor_FRONT;
  		WaitTime\InPos, 1;
		AG_FY_DEFLECTION := CRobT(\Tool:=tWeldGun\WObj:=obSTN1);
        WaitTime\InPos, 1;
        AG_FY_DEFLECTION.trans.y := AG_FY_DEFLECTION.trans.y - NOZZLE_RADIUS;
        WaitTime\InPos, 0.2;
        MoveL SP_AGFY_S, v500, z1, tWeldGun\WObj:=wobjHanchor_FRONT;
        MoveL SP_AHFY_S, v500, z1, tWeldGun\WObj:=wobjHanchor_FRONT;
		Search_1D SR_AHF_Y1\SearchStop:=AH_FY, SP_AHFY_S, SP_AHFY_E, v50, tWeldGun\WObj:=wobjHanchor_FRONT\SchSpeed:=10;
        TPWrite "SR_AHF_Y1 DEFLECTION:="\Pos:=SR_AHF_Y1.trans;
		Search_1D SR_AHF_Y2\SearchStop:=AH_FY, SP_AHFY_S, SP_AHFY_E, v50, tWeldGun\WObj:=wobjHanchor_FRONT\SchSpeed:=10;
  		TPWrite "SR_AHF_Y2 DEFLECTION:="\Pos:=SR_AHF_Y2.trans;
        MoveL AH_FY, v50, fine, tWeldGun\WObj:=wobjHanchor_FRONT;
  		WaitTime\InPos, 1;
		AH_FY_DEFLECTION := CRobT(\Tool:=tWeldGun\WObj:=obSTN1);
        WaitTime\InPos, 1;
        AH_FY_DEFLECTION.trans.y := AH_FY_DEFLECTION.trans.y - NOZZLE_RADIUS;
        WaitTime\InPos, 0.2;
	    ! POSSIBLY NEED TO ADD A "Y" DISPLACEMENT TO KEEP THE "Z" SEARCH ON THE NOZZLE
        SR_AHF_Y2.TRANS.Y := SR_AHF_Y1.TRANS.Y;
		PDispSet SR_AHF_Y2;
		MoveL Offs(SP_AHFY_S,0,50,0), v500, z1, tWeldGun\WObj:=wobjHanchor_FRONT;
        MoveJ Offs(SP_AHFZ_S,0,400,50), v500, z1, tWeldGun\WObj:=wobjHanchor_FRONT;
        MoveJ Offs(SP_AHFZ_S,0,100,50), v500, z1, tWeldGun\WObj:=wobjHanchor_FRONT;
		MoveL SP_AHFZ_S, v500, z1, tWeldGun\WObj:=wobjHanchor_FRONT;
        Search_1D SR_AHF_Z\SearchStop:=AH_FZ, SP_AHFZ_S, SP_AHFZ_E, v50, tWeldGun\WObj:=wobjHanchor_FRONT\SchSpeed:=10;
  		MoveL AH_FZ, v50, fine, tWeldGun\WObj:=wobjHanchor_FRONT;
        WaitTime\InPos, 1;
        AH_FZ_DEFLECTION := CRobT(\Tool:=tWeldGun\WObj:=obSTN1);
        WaitTime\InPos, 1;
        TPWrite "SR_AGF_Z DEFLECTION:="\Pos:=SR_AGF_Z.trans;
		MoveL SP_AHFZ_S, v200, z1, tWeldGun\WObj:=wobjHanchor_FRONT;
        ! ADDED X SEARCH
 		MoveL SP_AHFX_S, v500, z1, tWeldGun\WObj:=wobjHanchor_FRONT;
        Search_1D SR_AHF_X\SearchStop:=AH_X, SP_AHFX_S, SP_AHFX_E, v50, tWeldGun\WObj:=wobjHanchor_FRONT\SchSpeed:=10;
		MoveL SP_AHFZ_S, v200, z1, tWeldGun\WObj:=wobjHanchor_FRONT;
        ! POSSIBLY NEED TO ADD A "Y" DISPLACEMENT TO KEEP THE "Z" SEARCH ON THE NOZZLE
        SR_AGF_Y2.TRANS.Y := SR_AGF_Y1.TRANS.Y;
		PDispSet SR_AGF_Y2;
        MoveJ SP_AGFZ_S, v500, z1, tWeldGun\WObj:=wobjHanchor_FRONT;
		Search_1D SR_AGF_Z\SearchStop:=AG_FZ, SP_AGFZ_S, SP_AGFZ_E, v50, tWeldGun\WObj:=wobjHanchor_FRONT\SchSpeed:=10;
   		MoveL AG_FZ, v50, fine, tWeldGun\WObj:=wobjHanchor_FRONT;
        WaitTime\InPos, 1;
        AG_FZ_DEFLECTION := CRobT(\Tool:=tWeldGun\WObj:=obSTN1);
        WaitTime\InPos, 1;
        TPWrite "SR_AGF_Z DEFLECTION:="\Pos:=SR_AGF_Z.trans;
		MoveL SP_AGFZ_S, v500, z1, tWeldGun\WObj:=wobjHanchor_FRONT;
        !ADDED X SEARCH
 		MoveL SP_AGFX_S, v500, z1, tWeldGun\WObj:=wobjHanchor_FRONT;
        Search_1D SR_AGF_X\SearchStop:=AG_X, SP_AGFX_S, SP_AGFX_E, v50, tWeldGun\WObj:=wobjHanchor_FRONT\SchSpeed:=10;
		MoveL SP_AGFZ_S, v200, z1, tWeldGun\WObj:=wobjHanchor_FRONT;
        MoveL OFFS(SP_AGFZ_S,0,100,75), v500, z1, tWeldGun\WObj:=wobjHanchor_FRONT;
        MoveL OFFS(SP_AGFZ_S,0,600,75), v500, z1, tWeldGun\WObj:=wobjHanchor_FRONT;
        FRONT_ANCHOR_ROTATION_DEFLECTION  wobjHanchor_FRONT_H, AH_FY_DEFLECTION, AH_FY, AH_FZ_DEFLECTION, AH_FZ;
        FRONT_ANCHOR_ROTATION_DEFLECTION  wobjHanchor_FRONT_G, AG_FY_DEFLECTION, AG_FY, AG_FZ_DEFLECTION, AG_FZ;
        FRONT_ANCHOR_TRANS_DEFLECTION wobjHanchor_FRONT_G, AG_FY_DEFLECTION, AG_FZ_DEFLECTION, AG_FY, AG_FZ  ;
        FRONT_ANCHOR_TRANS_DEFLECTION wobjHanchor_FRONT_H, AH_FY_DEFLECTION, AH_FZ_DEFLECTION, AH_FY, AH_FZ  ;
        SET_ANCHOR_X AG_X;
        SET_ANCHOR_X AH_X;
        MoveJ Offs(AG406,150,300,50), v500, z1, tWeldGun\WObj:=wobjHanchor_FRONT_G;
		MoveL RelTool(AG406,0,0,-30), v500, z1, tWeldGun\WObj:=wobjHanchor_FRONT_G;
        ArcLStart AG406, v100, smHCYLANCH, wdHCYLANCH\Weave:=wvHCYLANCH, fine, tWeldGun\WObj:=wobjHanchor_FRONT_G\Track:=trHCYLANCHhiteonly;
		ArcL AG407, v100, smHCYLANCH, wdHCYLANCH\Weave:=wvHCYLANCH, z10, tWeldGun\WObj:=wobjHanchor_FRONT_G\Track:=trHCYLANCHhiteonly;
		ArcLEnd AG408, v100, smHCYLANCH, wdHCYLANCH\Weave:=wvHCYLANCH, z10, tWeldGun\WObj:=wobjHanchor_FRONT_G\Track:=trHCYLANCHhiteonly;
		MoveL RelTool(AG408,0,0,-10), v200, z1, tWeldGun\WObj:=wobjHanchor_FRONT_G;
		MoveL RelTool(AG406,0,0,-150), vExtMax, z1, tWeldGun\WObj:=wobjHanchor_FRONT_G;
		MoveL Offs(AG406,150,250,50), vExtMax, z1, tWeldGun\WObj:=wobjHanchor_FRONT_G;
		MoveJ Offs(AG420,150,350,50), vExtMax, z1, tWeldGun\WObj:=wobjHanchor_FRONT_G;
		MoveJ Offs(AG420,50,350,50), vExtMax, z1, tWeldGun\WObj:=wobjHanchor_FRONT_G;
  		MoveJ Offs(AG420,50,50,50), vExtMax, z1, tWeldGun\WObj:=wobjHanchor_FRONT_G;
    	MoveL RelTool(AG420,0,0,-15), vExtMax, fine, tWeldGun\WObj:=wobjHanchor_FRONT_G;
		ArcLStart AG420, v100, smHCYLANCH, wdHCYLANCH\Weave:=wvHCYLANCH, fine, tWeldGun\WObj:=wobjHanchor_FRONT_G\Track:=trHCYLANCHhiteonly;
		ArcL AG419, v100, smHCYLANCH, wdHCYLANCH\Weave:=wvHCYLANCH, z10, tWeldGun\WObj:=wobjHanchor_FRONT_G\Track:=trHCYLANCHhiteonly;
		ArcLEnd AG418, v100, smHCYLANCH, wdHCYLANCH\Weave:=wvHCYLANCH, z10, tWeldGun\WObj:=wobjHanchor_FRONT_G\Track:=trHCYLANCHhiteonly;
		MoveL RelTool(AG419,0,-15,-15), vExtMax, fine, tWeldGun\WObj:=wobjHanchor_FRONT_G;
		MoveL RelTool(AG420,0,-15,-15), vExtMax, fine, tWeldGun\WObj:=wobjHanchor_FRONT_G;
  		MoveJ Offs(AG420,50,75,50), vExtMax, z1, tWeldGun\WObj:=wobjHanchor_FRONT_G;
  		MoveJ Offs(AG420,150,350,50), vExtMax, z1, tWeldGun\WObj:=wobjHanchor_FRONT_G;
  		IF bAnchor_Lite = TRUE THEN
  			MoveJ Offs(AG408,150,350,50), vExtMax, z1, tWeldGun\WObj:=wobjHanchor_FRONT_G;
  			GOTO Short_Cut;
  		ENDIF
        MoveJ Offs(AG403,75,350,-25), vExtMax, z1, tWeldGun\WObj:=wobjHanchor_FRONT_G;
		MoveL Offs(AG403,25,25,-25), vExtMax, z1, tWeldGun\WObj:=wobjHanchor_FRONT_G;
		MoveL RelTool(AG403,0,0,-15), vExtMax, fine, tWeldGun\WObj:=wobjHanchor_FRONT_G;
		ArcLStart AG403, v100, smHCYLANCH, wdHCYLANCH\Weave:=wvHCYLANCH, fine, tWeldGun\WObj:=wobjHanchor_FRONT_G\Track:=trHCYLANCHhiteonly;
		ArcL AG404, v100, smHCYLANCH, wdHCYLANCH\Weave:=wvHCYLANCH, z10, tWeldGun\WObj:=wobjHanchor_FRONT_G\Track:=trHCYLANCHhiteonly;
		ArcLEnd AG405, v100, smHCYLANCH, wdHCYLANCH\Weave:=wvHCYLANCH, z10, tWeldGun\WObj:=wobjHanchor_FRONT_G\Track:=trHCYLANCHhiteonly;
		MoveL RelTool(AG403,0,0,-15), vExtMax, fine, tWeldGun\WObj:=wobjHanchor_FRONT_G;
		MoveL Offs(AG403,30,100,-25), vExtMax, fine, tWeldGun\WObj:=wobjHanchor_FRONT_G;
		MoveL Offs(AG403,75,200,-40), vExtMax, fine, tWeldGun\WObj:=wobjHanchor_FRONT_G;
		MoveL Offs(AG403,850,450,50), vExtMax, fine, tWeldGun\WObj:=wobjHanchor_FRONT_G;
		Short_Cut:
 		MoveJ Offs(AH407,-150,450,50), vExtMax, z1, tWeldGun\WObj:=wobjHanchor_FRONT_H;
 		MoveL RelTool(AH406,0,0,-20), v500, z1, tWeldGun\WObj:=wobjHanchor_FRONT_H;
        ArcLStart AH406, v100, smHCYLANCH, wdHCYLANCH\Weave:=wvHCYLANCH, fine, tWeldGun\WObj:=wobjHanchor_FRONT_H\Track:=trHCYLANCHhiteonly;
		ArcL AH407, v100, smHCYLANCH, wdHCYLANCH\Weave:=wvHCYLANCH, z10, tWeldGun\WObj:=wobjHanchor_FRONT_H\Track:=trHCYLANCHhiteonly;
		ArcLEnd AH408, v100, smHCYLANCH, wdHCYLANCH\Weave:=wvHCYLANCH, z10, tWeldGun\WObj:=wobjHanchor_FRONT_H\Track:=trHCYLANCHhiteonly;
		MoveL RelTool(AH408,0,0,-10), v200, z1, tWeldGun\WObj:=wobjHanchor_FRONT_H;
		MoveL RelTool(AH406,0,0,-150), vExtMax, z1, tWeldGun\WObj:=wobjHanchor_FRONT_H;
		MoveJ Offs(AH406,-150,250,50), vExtMax, z1, tWeldGun\WObj:=wobjHanchor_FRONT_H;
		MoveJ Offs(AH420,-150,250,50), vExtMax, z1, tWeldGun\WObj:=wobjHanchor_FRONT_H;
		MoveL RelTool(AH420,0,0,-15), vExtMax, fine, tWeldGun\WObj:=wobjHanchor_FRONT_H;
  		ArcLStart AH420, v100, smHCYLANCH, wdHCYLANCH\Weave:=wvHCYLANCH, fine, tWeldGun\WObj:=wobjHanchor_FRONT_H\Track:=trHCYLANCHhiteonly;
  		ArcL AH419, v100, smHCYLANCH, wdHCYLANCH\Weave:=wvHCYLANCH, z10, tWeldGun\WObj:=wobjHanchor_FRONT_H\Track:=trHCYLANCHhiteonly;
  		ArcLEnd AH418, v100, smHCYLANCH, wdHCYLANCH\Weave:=wvHCYLANCH, z10, tWeldGun\WObj:=wobjHanchor_FRONT_H\Track:=trHCYLANCHhiteonly;
		PDispOff;
		MoveL RelTool(AH419,0,10,-15), vExtMax, fine, tWeldGun\WObj:=wobjHanchor_FRONT_H;
		MoveL RelTool(AH420,0,0,-15), vExtMax, fine, tWeldGun\WObj:=wobjHanchor_FRONT_H;
  		MoveJ Offs(AH420,-100,250,0), vExtMax, z1, tWeldGun\WObj:=wobjHanchor_FRONT_H;
  		IF bAnchor_Lite = TRUE THEN
  			MoveJ Offs(AH408,-350,450,20), vExtMax, z1, tWeldGun\WObj:=wobjHanchor_FRONT_G;
  			GOTO Shorter_Cut;
  		ENDIF
  		MoveJ Offs(AH406,-100,250,0), vExtMax, z1, tWeldGun\WObj:=wobjHanchor_FRONT_H;
       	MoveL Offs(AH403,-50,350,-50), vExtMax, z1, tWeldGun\WObj:=wobjHanchor_FRONT_H;
		MoveL Offs(AH403,-25,25,-25), vExtMax, z1, tWeldGun\WObj:=wobjHanchor_FRONT_H;
		MoveL RelTool(AH403,0,0,-15), vExtMax, fine, tWeldGun\WObj:=wobjHanchor_FRONT_H;
		ArcLStart AH403, v100, smHCYLANCH, wdHCYLANCH\Weave:=wvHCYLANCH, fine, tWeldGun\WObj:=wobjHanchor_FRONT_H\Track:=trHCYLANCHhiteonly;
		ArcL AH404, v100, smHCYLANCH, wdHCYLANCH\Weave:=wvHCYLANCH, z10, tWeldGun\WObj:=wobjHanchor_FRONT_H\Track:=trHCYLANCHhiteonly;
		ArcLEnd AH405, v100, smHCYLANCH, wdHCYLANCH\Weave:=wvHCYLANCH, z10, tWeldGun\WObj:=wobjHanchor_FRONT_H\Track:=trHCYLANCHhiteonly;
		MoveL RelTool(AH403,0,0,-15), vExtMax, fine, tWeldGun\WObj:=wobjHanchor_FRONT_H;
		MoveL Offs(AH403,-50,50,-25), vExtMax, fine, tWeldGun\WObj:=wobjHanchor_FRONT_H;
		MoveL Offs(AH403,-100,150,-25), vExtMax, fine, tWeldGun\WObj:=wobjHanchor_FRONT_H;
		MoveL Offs(AH403,-250,250,-25), vExtMax, fine, tWeldGun\WObj:=wobjHanchor_FRONT_H;
		Shorter_Cut:
        MoveL Offs(AH408,-350,450,20), vExtMax, z1, tWeldGun\WObj:=wobjHanchor_FRONT_H;
        MoveJ pjthomeSTA1zero, vCellSpeed, fine, tWeldGun\WObj:=wobj0;
        LABEL:
    ENDPROC

    PROC WELD_AN_H_ANCHOR()
    !THE WOBJ WRINKLE HAS BEEN REMOVED FROM THIS PROC 08-09-17!!!!!!!!!!!
    !!!!!THIS PROGRAM IS now revised FOR H ANCHORS TO GET SEARCHED IN POSITION 11-29-17!!!!!!!
    !!!!! nozzle search version 12-27-17!!!!!!!!!!!
    !!!!!!!!!!!!!!!!REVISED 03-16-18 to add anchor_back X searches!!!!!
        ActUnit STN1;
		AccSet 40, 40;
        MoveJ pjthomeSTA1zero, vCellSpeed, fine, tWeldGun\WObj:=wobj0;
		MoveJ Offs(SP_AGBY_S,0,-100,50), v300, z5, tWeldGun\WObj:=wobjHanchor_BACK;
        MoveL SP_AGBY_S, v200, z5, tWeldGun\WObj:=wobjHanchor_BACK;
		Search_1D SR_AGB_Y\SearchStop:=AG_BY, SP_AGBY_S, SP_AGBY_E, v50, tWeldGun\WObj:=wobjHanchor_BACK\SchSpeed:=10;
  		MoveL AG_BY, v50, fine, tWeldGun\WObj:=wobjHanchor_BACK;
  		WaitTime\InPos, 1;
		AG_BY_DEFLECTION := CRobT(\Tool:=tWeldGun\WObj:=obSTN1);
        WaitTime\InPos, .2;
        AG_BY_DEFLECTION.trans.y := AG_BY_DEFLECTION.trans.y + NOZZLE_RADIUS;
        WaitTime\InPos, .2;
        TPWrite "SR_AGB_Y DEFLECTION:="\Pos:=SR_AGB_Y.trans;
		MoveL SP_AGBY_S, v300, z5, tWeldGun\WObj:=wobjHanchor_BACK;
        MoveL SP_AHBY_S, v50, z5, tWeldGun\WObj:=wobjHanchor_BACK;
		Search_1D SR_AHB_Y\SearchStop:=AH_BY, SP_AHBY_S, SP_AHBY_E, v50, tWeldGun\WObj:=wobjHanchor_BACK\SchSpeed:=10;
  		MoveL AH_BY, v50, fine, tWeldGun\WObj:=wobjHanchor_BACK;
  		WaitTime\InPos, 1;
		AH_BY_DEFLECTION := CRobT(\Tool:=tWeldGun\WObj:=obSTN1);
        WaitTime\InPos, .2;
        AH_BY_DEFLECTION.trans.y := AH_BY_DEFLECTION.trans.y + NOZZLE_RADIUS;
        WaitTime\InPos, .2;
			TPWrite "SR_AHB_Y DEFLECTION:="\Pos:=SR_AHB_Y.trans;
		MoveL SP_AHBY_S, v200, z5, tWeldGun\WObj:=wobjHanchor_BACK;
	    MoveJ Offs(SP_AHBY_S,0,-275,75), v100, z5, tWeldGun\WObj:=wobjHanchor_BACK;
	    MoveJ Offs(SP_AHBY_S,0,-325,125), v100, z5, tWeldGun\WObj:=wobjHanchor_BACK;
	    MoveL Offs(SP_AGBY_S,0,-325,125), v100, z5, tWeldGun\WObj:=wobjHanchor_BACK;
		MoveJ Offs(SP_GX_S,0,-50,125), v100, z5, tWeldGun\WObj:=wobjHanchor_BACK;
        MoveL SP_GX_S, v200, z1, tWeldGun\WObj:=wobjHanchor;
		Search_1D SR_AG_X\SearchStop:=AG_X, SP_GX_S, SP_GX_E, v50, tWeldGun\WObj:=wobjHanchor\SchSpeed:=10;
        TPWrite "SR_AG_X :="\Pos:=SR_AG_X.trans;
		MoveL SP_GX_S, v200, z1, tWeldGun\WObj:=wobjHanchor;
        MoveL SP_AGBZ_S, v200, z1, tWeldGun\WObj:=wobjHanchor_BACK;
	    Search_1D SR_AGB_Z\SearchStop:=AG_BZ, SP_AGBZ_S, SP_AGBZ_E, v50, tWeldGun\WObj:=wobjHanchor_BACK\SchSpeed:=10;
     	MoveL AG_BZ, v50, fine, tWeldGun\WObj:=wobjHanchor_BACK;
  		WaitTime\InPos, 1;
		AG_BZ_DEFLECTION := CRobT(\Tool:=tWeldGun\WObj:=obSTN1);
        WaitTime\InPos, 1;
        TPWrite "SR_AGB_Z DEFLECTION:="\Pos:=SR_AGB_Z.trans;
        MoveL SP_AGBZ_S, v200, z1, tWeldGun\WObj:=wobjHanchor_BACK;
        MoveL SP_AHBZ_S, v50, z1, tWeldGun\WObj:=wobjHanchor_BACK;
	    Search_1D SR_AHB_Z\SearchStop:=AH_BZ, SP_AHBZ_S, SP_AHBZ_E, v50, tWeldGun\WObj:=wobjHanchor_BACK\SchSpeed:=10;
     	MoveL AH_BZ, v50, fine, tWeldGun\WObj:=wobjHanchor_BACK;
  		WaitTime\InPos, 1;
		AH_BZ_DEFLECTION := CRobT(\Tool:=tWeldGun\WObj:=obSTN1);
        WaitTime\InPos, 1;
        TPWrite "SR_AHB_Z DEFLECTION:="\Pos:=SR_AHB_Z.trans;
        MoveL SP_AHBZ_S, v200, z1, tWeldGun\WObj:=wobjHanchor_BACK;
        MoveL SP_HX_S, v200, z1, tWeldGun\WObj:=wobjHanchor;
		Search_1D SR_AH_X\SearchStop:=AH_X, SP_HX_S, SP_HX_E, v50, tWeldGun\WObj:=wobjHanchor\SchSpeed:=10;
        TPWrite "SR_AH_X :="\Pos:=SR_AH_X.trans;
		MoveL SP_HX_S, v200, z1, tWeldGun\WObj:=wobjHanchor;
		MoveL Offs(SP_AHBZ_S,0,-125,50), v200, z5, tWeldGun\WObj:=wobjHanchor_BACK;
		MoveL Offs(SP_AHBZ_S,0,-500,100), v200, z5, tWeldGun\WObj:=wobjHanchor_BACK;
        RESET_ANCHOR_BACK_WOBJ;
        SET_ANCHOR_X AG_X;
        SET_ANCHOR_X AH_X;
        TPWrite "NOW WORKING ON WELD 'AH_BACK'";
		MoveJ Offs(AH301,-150,-250,-10), vExtMax, z1, tWeldGun\WObj:=wobjHanchor_BACK_H;
		MoveL RelTool(AH300,0,0,-20), v200, z1, tWeldGun\WObj:=wobjHanchor_BACK_H;
		ArcLStart AH300, v100, smHCYLANCH, wdHCYLANCH\Weave:=wvHCYLANCH, fine, tWeldGun\WObj:=wobjHanchor_BACK_H\Track:=trHCYLANCHhiteonly;
		ArcL AH301, v100, smHCYLANCH, wdHCYLANCH\Weave:=wvHCYLANCH, z10, tWeldGun\WObj:=wobjHanchor_BACK_H\Track:=trHCYLANCHhiteonly;
		IF bAnchor_Lite = TRUE THEN
			ArcLEnd AH302, v100, smHCYLANCH, wdHCYLANCH\Weave:=wvHCYLANCH, z10, tWeldGun\WObj:=wobjHanchor_BACK_H\Track:=trHCYLANCHhiteonly;
			GOTO Short_Cut;
		ENDIF
		ArcL AH302, v100, smHCYLANCH, wdHCYLANCH\Weave:=wvHCYLANCH, z10, tWeldGun\WObj:=wobjHanchor_BACK_H\Track:=trHCYLANCHhiteonly;
		ArcCEnd AH303, AH304, v100, smHCYLANCH, wdHCYLANCH\Weave:=wvHCYLANCH, z10, tWeldGun\WObj:=wobjHanchor_BACK_H\Track:=trHCYLANCHhiteonly;
		MoveL RelTool(AH304,0,0,-10), v200, z1, tWeldGun\WObj:=wobjHanchor_BACK_H;
		MoveL RelTool(AH303,0,0,-5), v200, z1, tWeldGun\WObj:=wobjHanchor_BACK_H;
		Short_Cut:
		MoveL RelTool(AH302,0,0,-100), v200, z1, tWeldGun\WObj:=wobjHanchor_BACK;
		MoveJ Offs(AH302,-50,-175,0), vExtMax, z1, tWeldGun\WObj:=wobjHanchor_BACK;
	    TPWrite "NOW WORKING ON WELD 'AG_BACK'";
		MoveL Offs(AG301,50,-150,0), vExtMax, z1, tWeldGun\WObj:=wobjHanchor_BACK;
		MoveL RelTool(AG300,0,0,-20), v200, z1, tWeldGun\WObj:=wobjHanchor_BACK;
		ArcLStart AG300, v100, smHCYLANCH, wdHCYLANCH\Weave:=wvHCYLANCH, fine, tWeldGun\WObj:=wobjHanchor_BACK_G\Track:=trHCYLANCHhiteonly;
		ArcL AG301, v100, smHCYLANCH, wdHCYLANCH\Weave:=wvHCYLANCH, z10, tWeldGun\WObj:=wobjHanchor_BACK_G\Track:=trHCYLANCHhiteonly;
		IF bAnchor_Lite = TRUE THEN
			ArcLEnd AG302, v100, smHCYLANCH, wdHCYLANCH\Weave:=wvHCYLANCH, z10, tWeldGun\WObj:=wobjHanchor_BACK_G\Track:=trHCYLANCHhiteonly;
			GOTO Shorter_Cut;
		ENDIF
		ArcL AG302, v100, smHCYLANCH, wdHCYLANCH\Weave:=wvHCYLANCH, z10, tWeldGun\WObj:=wobjHanchor_BACK_G\Track:=trHCYLANCHhiteonly;
		ArcCEnd AG303, AG304, v100, smHCYLANCH, wdHCYLANCH\Weave:=wvHCYLANCH, z10, tWeldGun\WObj:=wobjHanchor_BACK_G\Track:=trHCYLANCHhiteonly;
		MoveL RelTool(AG303,0,-50,-100), v200, z1, tWeldGun\WObj:=wobjHanchor_BACK;
		Shorter_Cut:
		MoveL Offs(AG302,300,-650,50), v200, z1, tWeldGun\WObj:=wobjHanchor_BACK;
		!CutWire;
		ActUnit STN1;
		MoveJ pjthomeSTA1zero, vCellSpeed, fine, tWeldGun\WObj:=wobj0;
        !!!!!!!!!!!  WILLIE MAKE IT   !!!!!!!!!!!
        MoveJ Offs(SP_AGFY_S,0,400,0), v1000, z5, tWeldGun\WObj:=wobjHanchor_FRONT;
        !!!!!!!!!!!  WILLIE MAKE IT   !!!!!!!!!!!
        MoveJ Offs(SP_AGFY_S,0,150,0), v400, z5, tWeldGun\WObj:=wobjHanchor_FRONT;
        MoveL SP_AGFY_S, v200, z1, tWeldGun\WObj:=wobjHanchor_FRONT;
		Search_1D SR_AGF_Y1\SearchStop:=AG_FY, SP_AGFY_S, SP_AGFY_E, v50, tWeldGun\WObj:=wobjHanchor_FRONT\SchSpeed:=10;
        TPWrite "SR_AGF_Y1 DEFLECTION:="\Pos:=SR_AGF_Y1.trans;
		Search_1D SR_AGF_Y2\SearchStop:=AG_FY, SP_AGFY_S, SP_AGFY_E, v50, tWeldGun\WObj:=wobjHanchor_FRONT\SchSpeed:=10;
        TPWrite "SR_AGF_Y2 DEFLECTION:="\Pos:=SR_AGF_Y2.trans;
        MoveL AG_FY, v50, fine, tWeldGun\WObj:=wobjHanchor_FRONT;
  		WaitTime\InPos, 1;
		AG_FY_DEFLECTION := CRobT(\Tool:=tWeldGun\WObj:=obSTN1);
        WaitTime\InPos, 1;
        AG_FY_DEFLECTION.trans.y := AG_FY_DEFLECTION.trans.y - NOZZLE_RADIUS;
        WaitTime\InPos, .2;
		MoveL SP_AGFY_S, v300, z1, tWeldGun\WObj:=wobjHanchor_FRONT;
        MoveL SP_AHFY_S, v50, z1, tWeldGun\WObj:=wobjHanchor_FRONT;
		Search_1D SR_AHF_Y1\SearchStop:=AH_FY, SP_AHFY_S, SP_AHFY_E, v50, tWeldGun\WObj:=wobjHanchor_FRONT\SchSpeed:=10;
        TPWrite "SR_AHF_Y1 DEFLECTION:="\Pos:=SR_AHF_Y1.trans;
		Search_1D SR_AHF_Y2\SearchStop:=AH_FY, SP_AHFY_S, SP_AHFY_E, v50, tWeldGun\WObj:=wobjHanchor_FRONT\SchSpeed:=10;
  		TPWrite "SR_AHF_Y2 DEFLECTION:="\Pos:=SR_AHF_Y2.trans;
        MoveL AH_FY, v50, fine, tWeldGun\WObj:=wobjHanchor_FRONT;
  		WaitTime\InPos, 1;
		AH_FY_DEFLECTION := CRobT(\Tool:=tWeldGun\WObj:=obSTN1);
        WaitTime\InPos, 1;
        AH_FY_DEFLECTION.trans.y := AH_FY_DEFLECTION.trans.y - NOZZLE_RADIUS;
        WaitTime\InPos, .2;
	    ! POSSIBLY NEED TO ADD A "Y" DISPLACEMENT TO KEEP THE "Z" SEARCH ON THE NOZZLE
        SR_AHF_Y2.TRANS.Y := SR_AHF_Y1.TRANS.Y;
		PDispSet SR_AHF_Y2;
		MoveJ Offs(SP_AHFY_S,0,300,0), v300, z1, tWeldGun\WObj:=wobjHanchor_FRONT;
		MoveJ [[45.40,353.50,-5.00],[0.117883,0.115262,-0.689484,0.705287],[-1,0,-1,0],[9E+09,0,135,9E+09,9E+09,9E+09]], v300, z1, tWeldGun\WObj:=wobjHanchor_FRONT;
        MoveJ Offs(SP_AHFZ_S,0,400,150), v300, z1, tWeldGun\WObj:=wobjHanchor_FRONT;
        MoveJ Offs(SP_AHFZ_S,0,100,50), v300, z1, tWeldGun\WObj:=wobjHanchor_FRONT;
		MoveL SP_AHFZ_S, v200, z1, tWeldGun\WObj:=wobjHanchor_FRONT;
        Search_1D SR_AHF_Z\SearchStop:=AH_FZ, SP_AHFZ_S, SP_AHFZ_E, v50, tWeldGun\WObj:=wobjHanchor_FRONT\SchSpeed:=10;
  		MoveL AH_FZ, v50, fine, tWeldGun\WObj:=wobjHanchor_FRONT;
        WaitTime\InPos, 1;
        AH_FZ_DEFLECTION := CRobT(\Tool:=tWeldGun\WObj:=obSTN1);
        WaitTime\InPos, 1;
        TPWrite "SR_AGF_Z DEFLECTION:="\Pos:=SR_AGF_Z.trans;
		MoveL SP_AHFZ_S, v200, z1, tWeldGun\WObj:=wobjHanchor_FRONT;
        !ADDED X SEARCH
  		MoveL SP_AHFX_S, v200, z1, tWeldGun\WObj:=wobjHanchor_FRONT;
        Search_1D SR_AHF_X\SearchStop:=AH_X, SP_AHFX_S, SP_AHFX_E, v50, tWeldGun\WObj:=wobjHanchor_FRONT\SchSpeed:=10;
		MoveL SP_AHFZ_S, v200, z1, tWeldGun\WObj:=wobjHanchor_FRONT;
        ! POSSIBLY NEED TO ADD A "Y" DISPLACEMENT TO KEEP THE "Z" SEARCH ON THE NOZZLE
        SR_AGF_Y2.TRANS.Y := SR_AGF_Y1.TRANS.Y;
		PDispSet SR_AGF_Y2;
        MoveL SP_AGFZ_S, v50, z1, tWeldGun\WObj:=wobjHanchor_FRONT;
		Search_1D SR_AGF_Z\SearchStop:=AG_FZ, SP_AGFZ_S, SP_AGFZ_E, v50, tWeldGun\WObj:=wobjHanchor_FRONT\SchSpeed:=10;
   		MoveL AG_FZ, v50, fine, tWeldGun\WObj:=wobjHanchor_FRONT;
        WaitTime\InPos, 1;
        AG_FZ_DEFLECTION := CRobT(\Tool:=tWeldGun\WObj:=obSTN1);
        WaitTime\InPos, 1;
        TPWrite "SR_AGF_Z DEFLECTION:="\Pos:=SR_AGF_Z.trans;
		MoveL SP_AGFZ_S, v200, z1, tWeldGun\WObj:=wobjHanchor_FRONT;
        !ADDED X SEARCH
  		MoveL SP_AGFX_S, v200, z1, tWeldGun\WObj:=wobjHanchor_FRONT;
        Search_1D SR_AGF_X\SearchStop:=AG_X, SP_AGFX_S, SP_AGFX_E, v50, tWeldGun\WObj:=wobjHanchor_FRONT\SchSpeed:=10;
		MoveL SP_AGFZ_S, v200, z1, tWeldGun\WObj:=wobjHanchor_FRONT;
        MoveL OFFS(SP_AGFZ_S,0,100,75), v200, z1, tWeldGun\WObj:=wobjHanchor_FRONT;
        MoveL OFFS(SP_AGFZ_S,0,600,75), v400, z1, tWeldGun\WObj:=wobjHanchor_FRONT;
        FRONT_ANCHOR_ROTATION_DEFLECTION  wobjHanchor_FRONT_H, AH_FY_DEFLECTION, AH_FY, AH_FZ_DEFLECTION, AH_FZ;
        FRONT_ANCHOR_ROTATION_DEFLECTION  wobjHanchor_FRONT_G, AG_FY_DEFLECTION, AG_FY, AG_FZ_DEFLECTION, AG_FZ;
        FRONT_ANCHOR_TRANS_DEFLECTION wobjHanchor_FRONT_G, AG_FY_DEFLECTION, AG_FZ_DEFLECTION, AG_FY, AG_FZ  ;
        FRONT_ANCHOR_TRANS_DEFLECTION wobjHanchor_FRONT_H, AH_FY_DEFLECTION, AH_FZ_DEFLECTION, AH_FY, AH_FZ  ;
        SET_ANCHOR_X  AG_X;
        SET_ANCHOR_X  AH_X;
        MoveJ Offs(AG306,150,300,50), v400, z1, tWeldGun\WObj:=wobjHanchor_FRONT_G;
		MoveL RelTool(AG306,0,0,-30), v200, z1, tWeldGun\WObj:=wobjHanchor_FRONT_G;
        ArcLStart AG306, v100, smHCYLANCH, wdHCYLANCH\Weave:=wvHCYLANCH, fine, tWeldGun\WObj:=wobjHanchor_FRONT_G\Track:=trHCYLANCHhiteonly;
		ArcL AG307, v100, smHCYLANCH, wdHCYLANCH\Weave:=wvHCYLANCH, z10, tWeldGun\WObj:=wobjHanchor_FRONT_G\Track:=trHCYLANCHhiteonly;
		IF bAnchor_Lite = TRUE THEN
			ArcLEnd AG308, v100, smHCYLANCH, wdHCYLANCH\Weave:=wvHCYLANCH, z10, tWeldGun\WObj:=wobjHanchor_FRONT_G\Track:=trHCYLANCHhiteonly;
			GOTO Shortest_Cut;
		ENDIF
		ArcL AG308, v100, smHCYLANCH, wdHCYLANCH\Weave:=wvHCYLANCH, z10, tWeldGun\WObj:=wobjHanchor_FRONT_G\Track:=trHCYLANCHhiteonly;
		ArcCEnd AG309, AG310, v100, smHCYLANCH, wdHCYLANCH\Weave:=wvHCYLANCH, z10, tWeldGun\WObj:=wobjHanchor_FRONT_G\Track:=trHCYLANCHhiteonly;
		MoveL RelTool(AG310,0,0,-10), v200, z1, tWeldGun\WObj:=wobjHanchor_FRONT_G;
		MoveL RelTool(AG309,0,0,-10), v200, z1, tWeldGun\WObj:=wobjHanchor_FRONT_G;
		Shortest_Cut:
		MoveL RelTool(AG306,0,0,-150), vExtMax, z1, tWeldGun\WObj:=wobjHanchor_FRONT_G;
		MoveL Offs(AG306,150,450,50), vExtMax, z1, tWeldGun\WObj:=wobjHanchor_FRONT_G;
   		MoveJ Offs(AH308,-150,450,50), vExtMax, z1, tWeldGun\WObj:=wobjHanchor_FRONT_H;
 		MoveL RelTool(AH306,0,0,-20), v200, z1, tWeldGun\WObj:=wobjHanchor_FRONT_H;
        ArcLStart AH306, v100, smHCYLANCH, wdHCYLANCH\Weave:=wvHCYLANCH, fine, tWeldGun\WObj:=wobjHanchor_FRONT_H\Track:=trHCYLANCHhiteonly;
		ArcL AH307, v100, smHCYLANCH, wdHCYLANCH\Weave:=wvHCYLANCH, z10, tWeldGun\WObj:=wobjHanchor_FRONT_H\Track:=trHCYLANCHhiteonly;
		IF bAnchor_Lite = TRUE THEN
			ArcLEnd AH308, v100, smHCYLANCH, wdHCYLANCH\Weave:=wvHCYLANCH, z10, tWeldGun\WObj:=wobjHanchor_FRONT_H\Track:=trHCYLANCHhiteonly;
			GOTO Cut_Off;
		ENDIF
		ArcL AH308, v100, smHCYLANCH, wdHCYLANCH\Weave:=wvHCYLANCH, z10, tWeldGun\WObj:=wobjHanchor_FRONT_H\Track:=trHCYLANCHhiteonly;
		ArcCEnd AH309, AH310, v100, smHCYLANCH, wdHCYLANCH\Weave:=wvHCYLANCH, z10, tWeldGun\WObj:=wobjHanchor_FRONT_H\Track:=trHCYLANCHhiteonly;
        MoveL RelTool(AH309,0,0,-10), v200, z1, tWeldGun\WObj:=wobjHanchor_FRONT_H;
        Cut_Off:
		MoveL RelTool(AH308,0,0,-75), vExtMax, z1, tWeldGun\WObj:=wobjHanchor_FRONT_H;
		MoveJ Offs(AH307,-150,300,50), vExtMax, z1, tWeldGun\WObj:=wobjHanchor_FRONT_H;
        MoveL Offs(AH307,-350,550,20), vExtMax, z1, tWeldGun\WObj:=wobjHanchor_FRONT_H;
        MoveJ pjthomeSTA1zero, vCellSpeed, fine, tWeldGun\WObj:=wobj0;
        LABEL:
    ENDPROC

    PROC WELD_AN_42H_ANCHOR()
    !!!!!THIS PROGRAM IS now revised FOR 42H ANCHORS TO GET SEARCHED IN POSITION 12-06-17!!!!!!!
    !!!!! nozzle search version (5.61 compatible) 01-29-17!!!!!!!!!!!
    !!!!!!!!!!!!!!!!REVISED 03-16-18 to add anchor_back X searches!!!!!
        ActUnit STN1;
		AccSet 40, 40;
        MoveJ pjthomeSTA1zero, vCellSpeed, fine, tWeldGun\WObj:=wobj0;
        MoveJ Offs(SP_AGBY_S,0,-300,50), v400, z5, tWeldGun\WObj:=wobjHanchor_BACK;
		MoveL Offs(SP_AGBY_S,0,-100,50), v300, z5, tWeldGun\WObj:=wobjHanchor_BACK;
        MoveL SP_AGBY_S, v200, z5, tWeldGun\WObj:=wobjHanchor_BACK;
		Search_1D SR_AGB_Y\SearchStop:=AG_BY, SP_AGBY_S, SP_AGBY_E, v50, tWeldGun\WObj:=wobjHanchor_BACK\SchSpeed:=10;
  		MoveL AG_BY, v50, fine, tWeldGun\WObj:=wobjHanchor_BACK;
  		WaitTime\InPos, 1;
		AG_BY_DEFLECTION := CRobT(\Tool:=tWeldGun\WObj:=obSTN1);
        WaitTime\InPos, 1;
        AG_BY_DEFLECTION.trans.y := AG_BY_DEFLECTION.trans.y + NOZZLE_RADIUS;
        WaitTime\InPos, 0.2;
        TPWrite "SR_AGB_Y DEFLECTION:="\Pos:=SR_AGB_Y.trans;
		MoveL SP_AGBY_S, v300, z5, tWeldGun\WObj:=wobjHanchor_BACK;
		MoveL Offs(SP_AGBY_S,0,-300,50), v300, z5, tWeldGun\WObj:=wobjHanchor_BACK;
		MoveJ Offs(SP_AHBY_S,0,-300,50), v300, z5, tWeldGun\WObj:=wobjHanchor_BACK;
        MoveL SP_AHBY_S, v300, z5, tWeldGun\WObj:=wobjHanchor_BACK;
		Search_1D SR_AHB_Y\SearchStop:=AH_BY, SP_AHBY_S, SP_AHBY_E, v50, tWeldGun\WObj:=wobjHanchor_BACK\SchSpeed:=10;
  		MoveL AH_BY, v50, fine, tWeldGun\WObj:=wobjHanchor_BACK;
  		WaitTime\InPos, 1;
		AH_BY_DEFLECTION := CRobT(\Tool:=tWeldGun\WObj:=obSTN1);
        WaitTime\InPos, 1;
        AH_BY_DEFLECTION.trans.y := AH_BY_DEFLECTION.trans.y + NOZZLE_RADIUS;
        WaitTime\InPos, 0.2;
		TPWrite "SR_AHB_Y DEFLECTION:="\Pos:=SR_AHB_Y.trans;
		MoveL SP_AHBY_S, v200, z5, tWeldGun\WObj:=wobjHanchor_BACK;
	    MoveJ Offs(SP_AHBY_S,0,-275,75), v100, z5, tWeldGun\WObj:=wobjHanchor_BACK;
	    MoveJ Offs(SP_AHBY_S,0,-325,125), v100, z5, tWeldGun\WObj:=wobjHanchor_BACK;
		MoveJ Offs(SP_GX_S,0,-250,125), v200, z5, tWeldGun\WObj:=wobjHanchor_BACK;
		MoveL Offs(SP_GX_S,0,-50,125), v200, z5, tWeldGun\WObj:=wobjHanchor_BACK;
        MoveL SP_GX_S, v200, z1, tWeldGun\WObj:=wobjHanchor;
		Search_1D SR_AG_X\SearchStop:=AG_X, SP_GX_S, SP_GX_E, v50, tWeldGun\WObj:=wobjHanchor\SchSpeed:=10;
        TPWrite "SR_AG_X :="\Pos:=SR_AG_X.trans;
		MoveL SP_GX_S, v200, z1, tWeldGun\WObj:=wobjHanchor;
        MoveL SP_AGBZ_S, v200, z1, tWeldGun\WObj:=wobjHanchor_BACK;
	    Search_1D SR_AGB_Z\SearchStop:=AG_BZ, SP_AGBZ_S, SP_AGBZ_E, v50, tWeldGun\WObj:=wobjHanchor_BACK\SchSpeed:=10;
     	MoveL AG_BZ, v50, fine, tWeldGun\WObj:=wobjHanchor_BACK;
  		WaitTime\InPos, 1;
		AG_BZ_DEFLECTION := CRobT(\Tool:=tWeldGun\WObj:=obSTN1);
        WaitTime\InPos, 1;
        TPWrite "SR_AGB_Z DEFLECTION:="\Pos:=SR_AGB_Z.trans;
        MoveL SP_AGBZ_S, v200, z1, tWeldGun\WObj:=wobjHanchor_BACK;
        MoveL Offs(SP_AGBZ_S,0,-225,100), v200, z1, tWeldGun\WObj:=wobjHanchor_BACK;
        MoveJ Offs(SP_AHBZ_S,0,-225,100), v200, z1, tWeldGun\WObj:=wobjHanchor_BACK;
        MoveL SP_AHBZ_S, v200, z1, tWeldGun\WObj:=wobjHanchor_BACK;
   	    Search_1D SR_AHB_Z\SearchStop:=AH_BZ, SP_AHBZ_S, SP_AHBZ_E, v50, tWeldGun\WObj:=wobjHanchor_BACK\SchSpeed:=10;
     	MoveL AH_BZ, v50, fine, tWeldGun\WObj:=wobjHanchor_BACK;
  		WaitTime\InPos, 1;
		AH_BZ_DEFLECTION := CRobT(\Tool:=tWeldGun\WObj:=obSTN1);
        WaitTime\InPos, 1;
        TPWrite "SR_AHB_Z DEFLECTION:="\Pos:=SR_AHB_Z.trans;
        MoveL SP_AHBZ_S, v200, z1, tWeldGun\WObj:=wobjHanchor_BACK;
        MoveL SP_HX_S, v200, z1, tWeldGun\WObj:=wobjHanchor;
		Search_1D SR_AH_X\SearchStop:=AH_X, SP_HX_S, SP_HX_E, v50, tWeldGun\WObj:=wobjHanchor\SchSpeed:=10;
        TPWrite "SR_AH_X :="\Pos:=SR_AH_X.trans;
		MoveL SP_HX_S, v200, z1, tWeldGun\WObj:=wobjHanchor;
		MoveL Offs(SP_AHBZ_S,0,-125,50), v200, z5, tWeldGun\WObj:=wobjHanchor_BACK;
		MoveL Offs(SP_AHBZ_S,0,-500,100), v200, z5, tWeldGun\WObj:=wobjHanchor_BACK;

        RESET_ANCHOR_BACK_WOBJ;
        SET_ANCHOR_X AG_X;
        SET_ANCHOR_X AH_X;

          TPWrite "NOW WORKING ON WELD 'AH_BACK'";
		MoveJ Offs(AH510,-150,-250,-10), vExtMax, z1, tWeldGun\WObj:=wobjHanchor_BACK_H;
		MoveL RelTool(AH511,0,0,-20), v200, z1, tWeldGun\WObj:=wobjHanchor_BACK_H;
		MoveL RelTool(AH511,0,0,-5), v200, z1, tWeldGun\WObj:=wobjHanchor_BACK_H;
   		ArcLStart AH511, v100, smHCYLANCH, wdHCYLANCH\Weave:=wvHCYLANCH, fine, tWeldGun\WObj:=wobjHanchor_BACK_H\Track:=trHCYLANCHhiteonly;
		ArcL AH510, v100, smHCYLANCH, wdHCYLANCH\Weave:=wvHCYLANCH, z10, tWeldGun\WObj:=wobjHanchor_BACK_H\Track:=trHCYLANCHhiteonly;
		ArcCEnd AH509,AH508, v100, smHCYLANCH, wdHCYLANCH\Weave:=wvHCYLANCH, z10, tWeldGun\WObj:=wobjHanchor_BACK_H\Track:=trHCYLANCHhiteonly;
		MoveL RelTool(AH508,0,0,-25), v200, z1, tWeldGun\WObj:=wobjHanchor_BACK_H;
		MoveL RelTool(AH509,0,0,-50), v200, z1, tWeldGun\WObj:=wobjHanchor_BACK_H;
		MoveL RelTool(AH510,0,0,-100), v200, z1, tWeldGun\WObj:=wobjHanchor_BACK_H;
            IF bAnchor_Lite = TRUE THEN
		    MoveL RelTool(AH512,0,0,-25), v200, z1, tWeldGun\WObj:=wobjHanchor_BACK_H;
            ArcLStart AH512, v100, smHCYLANCH, wdHCYLANCH\Weave:=wvHCYLANCH, fine, tWeldGun\WObj:=wobjHanchor_BACK_H\Track:=trHCYLANCHhiteonly;
	    	ArcLEnd AH513, v100, smHCYLANCH, wdHCYLANCH\Weave:=wvHCYLANCH, z10, tWeldGun\WObj:=wobjHanchor_BACK_H\Track:=trHCYLANCHhiteonly;
	    	MoveL RelTool(AH513,0,0,-25), v200, z1, tWeldGun\WObj:=wobjHanchor_BACK_H;
            GOTO Short_Cut;
		    ENDIF
        MoveL RelTool(AH512,0,0,-100), v200, z1, tWeldGun\WObj:=wobjHanchor_BACK_H;
        MoveL RelTool(AH512,0,0,-30), v200, z1, tWeldGun\WObj:=wobjHanchor_BACK_H;
		MoveL RelTool(AH512,0,0,-10), v200, z1, tWeldGun\WObj:=wobjHanchor_BACK_H;
        ArcLStart AH512, v100, smHCYLANCH, wdHCYLANCH\Weave:=wvHCYLANCH, fine, tWeldGun\WObj:=wobjHanchor_BACK_H\Track:=trHCYLANCHhiteonly;
		ArcL AH513, v100, smHCYLANCH, wdHCYLANCH\Weave:=wvHCYLANCH, z10, tWeldGun\WObj:=wobjHanchor_BACK_H\Track:=trHCYLANCHhiteonly;
		ArcCEnd AH514,AH515, v100, smHCYLANCH, wdHCYLANCH\Weave:=wvHCYLANCH, z10, tWeldGun\WObj:=wobjHanchor_BACK_H\Track:=trHCYLANCHhiteonly;
   		MoveL RelTool(AH515,0,0,-15), v200, z1, tWeldGun\WObj:=wobjHanchor_BACK_H;
		Short_Cut:
		MoveL RelTool(AH514,0,0,-100), v200, z1, tWeldGun\WObj:=wobjHanchor_BACK;
		MoveL Offs(AH512,-150,-450,0), vExtMax, z1, tWeldGun\WObj:=wobjHanchor_BACK;
        TPWrite "NOW WORKING ON WELD 'AG_BACK'";
		MoveJ Offs(AG511,150,-450,0), vExtMax, z1, tWeldGun\WObj:=wobjHanchor_BACK;
		MoveL RelTool(AG511,0,0,-120), v200, z1, tWeldGun\WObj:=wobjHanchor_BACK;
		MoveL RelTool(AG511,0,0,-20), v200, z1, tWeldGun\WObj:=wobjHanchor_BACK;
		ArcLStart AG511, v100, smHCYLANCH, wdHCYLANCH\Weave:=wvHCYLANCH, fine, tWeldGun\WObj:=wobjHanchor_BACK_H\Track:=trHCYLANCHhiteonly;
		ArcL AG510, v100, smHCYLANCH, wdHCYLANCH\Weave:=wvHCYLANCH, z10, tWeldGun\WObj:=wobjHanchor_BACK_H\Track:=trHCYLANCHhiteonly;
		ArcCEnd AG509,AG508, v100, smHCYLANCH, wdHCYLANCH\Weave:=wvHCYLANCH, z10, tWeldGun\WObj:=wobjHanchor_BACK_H\Track:=trHCYLANCHhiteonly;
   		MoveL RelTool(AG508,0,20,-25), v200, z1, tWeldGun\WObj:=wobjHanchor_BACK_H;
		MoveL RelTool(AG509,0,0,-100), v200, z1, tWeldGun\WObj:=wobjHanchor_BACK_H;
		MoveJ Offs(AG511,50,-150,0), v200, z1, tWeldGun\WObj:=wobjHanchor_BACK_H;
		!MoveJ pjthomeSTA1zero, vCellSpeed, fine, tWeldGun\WObj:=wobj0;
		MoveJ Offs(AG512,50,-150,0), v500, z1, tWeldGun\WObj:=wobjHanchor_BACK_H;
		IF bAnchor_Lite = TRUE THEN
		    MoveL RelTool(AG512,0,0,-25), v200, z1, tWeldGun\WObj:=wobjHanchor_BACK_H;
            ArcLStart AG512, v100, smHCYLANCH, wdHCYLANCH\Weave:=wvHCYLANCH, fine, tWeldGun\WObj:=wobjHanchor_BACK_G\Track:=trHCYLANCHhiteonly;
	    	ArcLEnd AG513, v100, smHCYLANCH, wdHCYLANCH\Weave:=wvHCYLANCH, z10, tWeldGun\WObj:=wobjHanchor_BACK_G\Track:=trHCYLANCHhiteonly;
	    	MoveL RelTool(AG513,0,0,-25), v200, z1, tWeldGun\WObj:=wobjHanchor_BACK_G;
            GOTO skip_it;
	  ENDIF
        MoveL RelTool(AG512,0,0,-10), v200, z1, tWeldGun\WObj:=wobjHanchor_BACK_G;
		ArcLStart AG512, v100, smHCYLANCH, wdHCYLANCH\Weave:=wvHCYLANCH, fine, tWeldGun\WObj:=wobjHanchor_BACK_H\Track:=trHCYLANCHhiteonly;
		ArcL AG513, v100, smHCYLANCH, wdHCYLANCH\Weave:=wvHCYLANCH, z10, tWeldGun\WObj:=wobjHanchor_BACK_H\Track:=trHCYLANCHhiteonly;
		ArcCEnd AG514,AG515, v100, smHCYLANCH, wdHCYLANCH\Weave:=wvHCYLANCH, z10, tWeldGun\WObj:=wobjHanchor_BACK_H\Track:=trHCYLANCHhiteonly;
   		MoveL RelTool(AG515,0,0,-25), v200, z1, tWeldGun\WObj:=wobjHanchor_BACK_G;
		MoveL RelTool(AG514,0,0,-50), v200, z1, tWeldGun\WObj:=wobjHanchor_BACK_G;
		MoveL RelTool(AG513,0,0,-65), v200, z1, tWeldGun\WObj:=wobjHanchor_BACK_G;
		skip_it:
		MoveJ Offs(AG512,50,-250,0), vExtMax, z1, tWeldGun\WObj:=wobjHanchor_BACK;
		MoveJ Offs(AG512,250,-450,0), vExtMax, z1, tWeldGun\WObj:=wobjHanchor_BACK;
		MoveJ pjthomeSTA1zero, vCellSpeed, fine, tWeldGun\WObj:=wobj0;
        !CutWire;
        ActUnit STN1;
        !!!!!!!!!!!  WILLIE MAKE IT   !!!!!!!!!!!
        MoveJ Offs(SP_AGFY_S,0,800,0), v1000, z5, tWeldGun\WObj:=wobjHanchor_FRONT;
        !!!!!!!!!!!  WILLIE MAKE IT   !!!!!!!!!!!
        !Stop;
        MoveJ Offs(SP_AGFY_S,0,150,0), v400, z5, tWeldGun\WObj:=wobjHanchor_FRONT;
        MoveL SP_AGFY_S, v200, z1, tWeldGun\WObj:=wobjHanchor_FRONT;
		Search_1D SR_AGF_Y1\SearchStop:=AG_FY, SP_AGFY_S, SP_AGFY_E, v50, tWeldGun\WObj:=wobjHanchor_FRONT\SchSpeed:=10;
        TPWrite "SR_AGF_Y1 DEFLECTION:="\Pos:=SR_AGF_Y1.trans;
		Search_1D SR_AGF_Y2\SearchStop:=AG_FY, SP_AGFY_S, SP_AGFY_E, v50, tWeldGun\WObj:=wobjHanchor_FRONT\SchSpeed:=10;
        TPWrite "SR_AGF_Y2 DEFLECTION:="\Pos:=SR_AGF_Y2.trans;
        MoveL AG_FY, v50, fine, tWeldGun\WObj:=wobjHanchor_FRONT;
  		WaitTime\InPos, 1;
		AG_FY_DEFLECTION := CRobT(\Tool:=tWeldGun\WObj:=obSTN1);
        WaitTime\InPos, 1;
        AG_FY_DEFLECTION.trans.y := AG_FY_DEFLECTION.trans.y - NOZZLE_RADIUS;
        WaitTime\InPos, 0.2;
 		MoveL SP_AGFY_S, v300, z1, tWeldGun\WObj:=wobjHanchor_FRONT;
        MoveL SP_AHFY_S, v300, z1, tWeldGun\WObj:=wobjHanchor_FRONT;
		Search_1D SR_AHF_Y1\SearchStop:=AH_FY, SP_AHFY_S, SP_AHFY_E, v50, tWeldGun\WObj:=wobjHanchor_FRONT\SchSpeed:=10;
        TPWrite "SR_AHF_Y1 DEFLECTION:="\Pos:=SR_AHF_Y1.trans;
		Search_1D SR_AHF_Y2\SearchStop:=AH_FY, SP_AHFY_S, SP_AHFY_E, v50, tWeldGun\WObj:=wobjHanchor_FRONT\SchSpeed:=10;
  		TPWrite "SR_AHF_Y2 DEFLECTION:="\Pos:=SR_AHF_Y2.trans;
        MoveL AH_FY, v50, fine, tWeldGun\WObj:=wobjHanchor_FRONT;
		AH_FY_DEFLECTION := CRobT(\Tool:=tWeldGun\WObj:=obSTN1);
        WaitTime\InPos, 1;
        AH_FY_DEFLECTION.trans.y := AH_FY_DEFLECTION.trans.y - NOZZLE_RADIUS;
        WaitTime\InPos, 1;
	    ! POSSIBLY NEED TO ADD A "Y" DISPLACEMENT TO KEEP THE "Z" SEARCH ON THE NOZZLE
        SR_AHF_Y2.TRANS.Y := SR_AHF_Y1.TRANS.Y;
		PDispSet SR_AHF_Y2;
		MoveL Offs(SP_AHFY_S,0,500,0), v300, z1, tWeldGun\WObj:=wobjHanchor_FRONT;
        MoveJ Offs(SP_AHFZ_S,0,400,150), v300, z1, tWeldGun\WObj:=wobjHanchor_FRONT;
        MoveJ Offs(SP_AHFZ_S,0,100,50), v300, z1, tWeldGun\WObj:=wobjHanchor_FRONT;
		MoveL SP_AHFZ_S, v200, z1, tWeldGun\WObj:=wobjHanchor_FRONT;
        Search_1D SR_AHF_Z\SearchStop:=AH_FZ, SP_AHFZ_S, SP_AHFZ_E, v50, tWeldGun\WObj:=wobjHanchor_FRONT\SchSpeed:=10;
  		MoveL AH_FZ, v50, fine, tWeldGun\WObj:=wobjHanchor_FRONT;
        WaitTime\InPos, 1;
        AH_FZ_DEFLECTION := CRobT(\Tool:=tWeldGun\WObj:=obSTN1);
        WaitTime\InPos, 1;
        TPWrite "SR_AGF_Z DEFLECTION:="\Pos:=SR_AGF_Z.trans;
		MoveL SP_AHFZ_S, v200, z1, tWeldGun\WObj:=wobjHanchor_FRONT;

        !ADDED X SEARCH
   		MoveL SP_AHFX_S, v200, z1, tWeldGun\WObj:=wobjHanchor_FRONT;
        Search_1D SR_AHF_X\SearchStop:=AH_X, SP_AHFX_S, SP_AHFX_E, v50, tWeldGun\WObj:=wobjHanchor_FRONT\SchSpeed:=10;
		MoveL SP_AHFZ_S, v200, z1, tWeldGun\WObj:=wobjHanchor_FRONT;

        MoveL Offs(SP_AHFZ_S,0,200,100), v200, z1, tWeldGun\WObj:=wobjHanchor_FRONT;
		MoveL Offs(SP_AGFZ_S,0,200,100), v200, z1, tWeldGun\WObj:=wobjHanchor_FRONT;
        ! POSSIBLY NEED TO ADD A "Y" DISPLACEMENT TO KEEP THE "Z" SEARCH ON THE NOZZLE
        SR_AGF_Y2.TRANS.Y := SR_AGF_Y1.TRANS.Y;
		PDispSet SR_AGF_Y2;
        MoveL SP_AGFZ_S, v200, z1, tWeldGun\WObj:=wobjHanchor_FRONT;
		Search_1D SR_AGF_Z\SearchStop:=AG_FZ, SP_AGFZ_S, SP_AGFZ_E, v50, tWeldGun\WObj:=wobjHanchor_FRONT\SchSpeed:=10;
   		MoveL AG_FZ, v50, fine, tWeldGun\WObj:=wobjHanchor_FRONT;
        WaitTime\InPos, 1;
        AG_FZ_DEFLECTION := CRobT(\Tool:=tWeldGun\WObj:=obSTN1);
        WaitTime\InPos, 1;
        TPWrite "SR_AGF_Z DEFLECTION:="\Pos:=SR_AGF_Z.trans;
		MoveL SP_AGFZ_S, v200, z1, tWeldGun\WObj:=wobjHanchor_FRONT;

        !ADDED X SEARCH
  		MoveL SP_AGFX_S, v200, z1, tWeldGun\WObj:=wobjHanchor_FRONT;
        Search_1D SR_AGF_X\SearchStop:=AG_X, SP_AGFX_S, SP_AGFX_E, v50, tWeldGun\WObj:=wobjHanchor_FRONT\SchSpeed:=10;
		MoveL SP_AGFZ_S, v200, z1, tWeldGun\WObj:=wobjHanchor_FRONT;

        MoveL OFFS(SP_AGFZ_S,0,100,75), v200, z1, tWeldGun\WObj:=wobjHanchor_FRONT;
        MoveL OFFS(SP_AGFZ_S,0,600,75), v400, z1, tWeldGun\WObj:=wobjHanchor_FRONT;
        FRONT_ANCHOR_ROTATION_DEFLECTION  wobjHanchor_FRONT_H, AH_FY_DEFLECTION, AH_FY, AH_FZ_DEFLECTION, AH_FZ;
        FRONT_ANCHOR_ROTATION_DEFLECTION  wobjHanchor_FRONT_G, AG_FY_DEFLECTION, AG_FY, AG_FZ_DEFLECTION, AG_FZ;
        FRONT_ANCHOR_TRANS_DEFLECTION wobjHanchor_FRONT_G, AG_FY_DEFLECTION, AG_FZ_DEFLECTION, AG_FY, AG_FZ  ;
        FRONT_ANCHOR_TRANS_DEFLECTION wobjHanchor_FRONT_H, AH_FY_DEFLECTION, AH_FZ_DEFLECTION, AH_FY, AH_FZ  ;
        SET_ANCHOR_X AG_X;
        SET_ANCHOR_X AH_X;

   		MoveJ Offs(AG501,150,300,50), v400, z1, tWeldGun\WObj:=wobjHanchor_FRONT_G;
		MoveJ RelTool(AG500,0,0,-30), v200, z1, tWeldGun\WObj:=wobjHanchor_FRONT_G;
        ArcLStart AG500, v100, smHCYLANCH, wdHCYLANCH\Weave:=wvHCYLANCH, fine, tWeldGun\WObj:=wobjHanchor_FRONT_G\Track:=trHCYLANCHhiteonly;
		ArcL AG501, v100, smHCYLANCH, wdHCYLANCH\Weave:=wvHCYLANCH, z10, tWeldGun\WObj:=wobjHanchor_FRONT_G\Track:=trHCYLANCHhiteonly;
		ArcCEnd AG502, AG503, v100, smHCYLANCH, wdHCYLANCH\Weave:=wvHCYLANCH, z10, tWeldGun\WObj:=wobjHanchor_FRONT_G\Track:=trHCYLANCHhiteonly;
		MoveL RelTool(AG502,0,0,-20), v200, z1, tWeldGun\WObj:=wobjHanchor_FRONT_G;
		MoveL Offs(AG501,30,50,0), v200, z1, tWeldGun\WObj:=wobjHanchor_FRONT_G;
		MoveL Offs(AG501,130,150,0), v200, z1, tWeldGun\WObj:=wobjHanchor_FRONT_G;
		MoveJ Offs(AG504,30,50,0), vExtMax, z1, tWeldGun\WObj:=wobjHanchor_FRONT_G;
 		MoveL RelTool(AG504,0,0,-20), v200, z1, tWeldGun\WObj:=wobjHanchor_FRONT_G;
        ArcLStart AG504, v100, smHCYLANCH, wdHCYLANCH\Weave:=wvHCYLANCH, fine, tWeldGun\WObj:=wobjHanchor_FRONT_G\Track:=trHCYLANCHhiteonly;
		IF bAnchor_Lite = TRUE THEN
			ArcLEnd AG505, v100, smHCYLANCH, wdHCYLANCH\Weave:=wvHCYLANCH, z10, tWeldGun\WObj:=wobjHanchor_FRONT_G\Track:=trHCYLANCHhiteonly;
			GOTO SKIP_THIS_WELD;
		ENDIF
		ArcL AG505, v100, smHCYLANCH, wdHCYLANCH\Weave:=wvHCYLANCH, z10, tWeldGun\WObj:=wobjHanchor_FRONT_G\Track:=trHCYLANCHhiteonly;
		ArcCEnd AG506, AG507, v100, smHCYLANCH, wdHCYLANCH\Weave:=wvHCYLANCH, z10, tWeldGun\WObj:=wobjHanchor_FRONT_G\Track:=trHCYLANCHhiteonly;
        MoveL RelTool(AG506,0,0,-10), v200, z1, tWeldGun\WObj:=wobjHanchor_FRONT_G;
        SKIP_THIS_WELD:
		MoveL RelTool(AG505,0,0,-75), vExtMax, z1, tWeldGun\WObj:=wobjHanchor_FRONT_G;
		MoveJ Offs(AG505,150,300,0), vExtMax, z1, tWeldGun\WObj:=wobjHanchor_FRONT_G;
        MoveJ Offs(AH505,-150,550,0), vExtMax, z1, tWeldGun\WObj:=wobjHanchor_FRONT_H;
        MoveJ Offs(AH501,-150,300,50), v400, z1, tWeldGun\WObj:=wobjHanchor_FRONT_H;
		MoveL RelTool(AH500,0,0,-30), v200, z1, tWeldGun\WObj:=wobjHanchor_FRONT_H;
        ArcLStart AH500, v100, smHCYLANCH, wdHCYLANCH\Weave:=wvHCYLANCH, fine, tWeldGun\WObj:=wobjHanchor_FRONT_H\Track:=trHCYLANCHhiteonly;
		ArcL AH501, v100, smHCYLANCH, wdHCYLANCH\Weave:=wvHCYLANCH, z10, tWeldGun\WObj:=wobjHanchor_FRONT_H\Track:=trHCYLANCHhiteonly;
		ArcCEnd AH502, AH503, v100, smHCYLANCH, wdHCYLANCH\Weave:=wvHCYLANCH, z10, tWeldGun\WObj:=wobjHanchor_FRONT_H\Track:=trHCYLANCHhiteonly;
		MoveL RelTool(AH502,0,0,-10), v200, z1, tWeldGun\WObj:=wobjHanchor_FRONT_H;
		MoveL RelTool(AH501,0,0,-35), v200, z1, tWeldGun\WObj:=wobjHanchor_FRONT_H;
		MoveL RelTool(AH505,0,0,-35), vExtMax, z1, tWeldGun\WObj:=wobjHanchor_FRONT_H;
 		MoveL RelTool(AH504,0,0,-20), v200, z1, tWeldGun\WObj:=wobjHanchor_FRONT_H;
        ArcLStart AH504, v100, smHCYLANCH, wdHCYLANCH\Weave:=wvHCYLANCH, fine, tWeldGun\WObj:=wobjHanchor_FRONT_H\Track:=trHCYLANCHhiteonly;
		IF bAnchor_Lite = TRUE THEN
			ArcLEnd AH505, v100, smHCYLANCH, wdHCYLANCH\Weave:=wvHCYLANCH, z10, tWeldGun\WObj:=wobjHanchor_FRONT_H\Track:=trHCYLANCHhiteonly;
			GOTO DONT_WELD_HERE;
		ENDIF
		ArcL AH505, v100, smHCYLANCH, wdHCYLANCH\Weave:=wvHCYLANCH, z10, tWeldGun\WObj:=wobjHanchor_FRONT_H\Track:=trHCYLANCHhiteonly;
		ArcCEnd AH506, AH507, v100, smHCYLANCH, wdHCYLANCH\Weave:=wvHCYLANCH, z10, tWeldGun\WObj:=wobjHanchor_FRONT_H\Track:=trHCYLANCHhiteonly;
        MoveL RelTool(AH507,0,0,-20), v200, z1, tWeldGun\WObj:=wobjHanchor_FRONT_H;
        MoveL RelTool(AH506,0,0,-50), v200, z1, tWeldGun\WObj:=wobjHanchor_FRONT_H;
        DONT_WELD_HERE:
		MoveL RelTool(AH505,0,0,-75), vExtMax, z1, tWeldGun\WObj:=wobjHanchor_FRONT_H;
		MoveJ Offs(AH505,-150,300,50), vExtMax, z1, tWeldGun\WObj:=wobjHanchor_FRONT_H;
        MoveL Offs(AH505,-350,550,20), vExtMax, z1, tWeldGun\WObj:=wobjHanchor_FRONT_H;
        MoveJ pjthomeSTA1zero, vCellSpeed, fine, tWeldGun\WObj:=wobj0;
        LABEL:

    ENDPROC
!!!!!!!!!!!!!!!!!!!!!!!!!!!!!!!!!!!!!!!!!!!!!!!!!!!!

    PROC WELD_THE_ANCHOR(
 INOUT
  num yy_of_search,
  num zz_of_search)
	VAR NUM ARM_WIDTH;

           IF PIVOT_USED =  674961 or PIVOT_USED =  350404 THEN  !77F - 120F CAM
                   ARM_WIDTH := (292/2) + SIDEPLATE + NOZZLE_RADIUS ;
           ELSEIF PIVOT_USED =  6099018 THEN  !18H CAM
                   ARM_WIDTH := (190.6/2) + SIDEPLATE + NOZZLE_RADIUS;
           ELSEIF PIVOT_USED =  6089330 THEN  !33H RND
                   ARM_WIDTH := (268/2) + NOZZLE_RADIUS ;
           ELSEIF PIVOT_USED =  6802774 THEN  !24H RND
                   ARM_WIDTH := (215.0/2) + NOZZLE_RADIUS ;
           ELSEIF PIVOT_USED =  6870131 THEN  !34H RND
                   ARM_WIDTH := (279.0/2) + NOZZLE_RADIUS ;
           ELSEIF  PIVOT_USED = 6845931 THEN  !42H
                   ARM_WIDTH := (287.0/2) + NOZZLE_RADIUS ;

           ENDIF

        ARM_G_XS.trans.x := (ARM_WIDTH + 60) * (-1);
		ARM_G_XS.trans.y := yy_of_search + 50;
		ARM_G_XS.trans.z := abs(zz_of_search);

		ARM_G_XE.trans.x := ARM_WIDTH * (-1);
		ARM_G_XE.trans.y := yy_of_search + 50;
		ARM_G_XE.trans.z := abs(zz_of_search);

		ARM_H_XS.trans.x := ARM_WIDTH + 60;
		ARM_H_XS.trans.y := yy_of_search + 50;
		ARM_H_XS.trans.z := abs(zz_of_search);

		ARM_H_XE.trans.x := ARM_WIDTH ;
		ARM_H_XE.trans.y := yy_of_search + 50;
		ARM_H_XE.trans.z := abs(zz_of_search);


        ActUnit STN1;
		AccSet 75, 75;
		MoveJ pjthomeSTA1zero, vCellSpeed, fine, tWeldGun\WObj:=wobj0;

        MoveJ offs(ARM_G_XS,-50,-500,0), vExtMax, fine, tWeldGun\WObj:=wobjHsideplate;
        MoveJ offs(ARM_G_XS,-50,0,0), vExtMax, fine, tWeldGun\WObj:=wobjHsideplate;
	    Search_1D ARM_G_X\SearchStop:=FAMILY_GX, ARM_G_XS, ARM_G_XE, v100, tWeldGun\WObj:=wobjHsideplate\SchSpeed:=10;
	    MoveJ offs(ARM_G_XS,-50,0,0), vExtMax, fine, tWeldGun\WObj:=wobjHsideplate;

        MoveJ offs(ARM_G_XS,-50,-500,0), vExtMax, fine, tWeldGun\WObj:=wobjHsideplate;
        MoveJ offs(ARM_H_XS,50,-500,0), vExtMax, fine, tWeldGun\WObj:=wobjHsideplate;

        MoveJ offs(ARM_H_XS,50,0,0), vExtMax, fine, tWeldGun\WObj:=wobjHsideplate;
		Search_1D ARM_H_X\SearchStop:=FAMILY_HX, ARM_H_XS, ARM_H_XE, v100, tWeldGun\WObj:=wobjHsideplate\SchSpeed:=10;
        MoveJ offs(ARM_H_XS,50,0,0), vExtMax, fine, tWeldGun\WObj:=wobjHsideplate;
        MoveJ offs(ARM_H_XS,50,-700,0), vExtMax, fine, tWeldGun\WObj:=wobjHsideplate;
		MoveJ pjthomeSTA1zero, vCellSpeed, fine, tWeldGun\WObj:=wobj0;
		The_Anchor_Lottery:

        INITIALIZE_DA_ANCHOR;

        IF ANCHOR_USED = 6089394 OR ANCHOR_USED = 6802707 THEN
               WELD_AN_H_ANCHOR;
        ELSEIF ANCHOR_USED = 6862141 THEN
               WELD_AN_42H_ANCHOR;
        ELSEIF  ANCHOR_USED = 689234 OR ANCHOR_USED = 6099135 OR ANCHOR_USED = 689899 THEN
               WELD_A_SQUARE_ANCHOR;
        ELSEIF ANCHOR_USED = 6850291 THEN
               WELD_A_TAPERED_SQUARE_ANCHOR;
        ENDIF

ANOTHERLABEL:

    ENDPROC

   PROC INITIALIZE_DA_ANCHOR()

   	        wobjHanchor_FRONT_G := wobjHanchor;
            wobjHanchor_FRONT_H := wobjHanchor;
            wobjHanchor_FRONT := wobjHanchor;
            FRAME_ANCHOR_FRONT_H := FRAME_ANCHOR   ;
            FRAME_ANCHOR_FRONT_G := FRAME_ANCHOR   ;
            FRAME_ANCHOR_FRONT := FRAME_ANCHOR   ;
            SET_ANCHOR_BACK_WOBJ;
            SET_ANCHOR_SRCH;
           IF bZEROING = TRUE THEN
        TPWrite ".............";
        TPWrite "THIS IS A FIRST PART EDIT";
        TPWrite "TURN OFF X IN JOG WINDOW";
        TPWrite "DO NOT EDIT FOR X";
        TPWrite "EDITING X WILL NOT WORK RIGHT";
        Stop;
        Stop;
        ELSEIF bZEROING = FALSE THEN
               GOTO EVERYPART;
        ENDIF
 EVERYPART:

   ENDPROC

  PROC Load_6806128R4()
!!!!!!!!!!!!!sk-32886!!!!!!!!!!!!!!!!!!!!!!!!!!!!!!!
   STICK_OUT := 2 ;
   SIDEPLATE := 12 ;
   FRONT_WRAPPER_THK := 8 ;
   BACK_WRAPPER_THK := 8 ;
   TIP_USED:= 6800124;
   ANCHOR_USED:=6099135;
   PIVOT_USED:= 6099018;
   b18H := TRUE;
   SEARCH_LENGTH := 35;
   bAnchor_Lite:=FALSE;
    !LOAD VARIABLES BELOW THIS LINE.
WANCHORANGLE:=86;
WANCHORX:=473.7;
WANCHORY:=199.3;
WOTOX:=928.7;
WPIVOTANGLE:=24;
WTIPANGLE:=21.5;
AA0:=0.5;
AA15:=-8.5;
AA18:=-17.5;
AA19:=-18.5;
AA21:=-0.5;
AA25:=12.5;
AA29:=23;
AA30:=11.5;
AA32:=0.5;
AA33:=-9.5;
AA34:=-11;
AA36:=-22.5;
AA38:=-34;
AA39:=-34;
AA41:=1.5;
AA42:=6.5;
AA45:=11.5;
AA46:=12.5;
AA47:=16.5;
AA48:=21.5;
AA49:=23;
AA61:=-11.5;
AA67:=-12.5;
AA69:=-13.5;
YY0:=-162.7;
YY15:=-155.3;
YY18:=-133.4;
YY19:=-128.8;
YY21:=-162.6;
YY25:=-147.4;
YY29:=-102.9;
YY30:=-277.3;
YY32:=-285.9;
YY33:=-280.2;
YY34:=-278.2;
YY36:=-254.7;
YY38:=-216.2;
YY39:=-184.6;
YY41:=-170.4;
YY42:=-166.4;
YY45:=-157.6;
YY46:=-155.3;
YY47:=-144.2;
YY48:=-126.3;
YY49:=-118.6;
YY61:=-157.8;
YY67:=-155.6;
YY69:=-152.8;
ZZ0:=-449.5;
ZZ15:=-352.3;
ZZ18:=-257.3;
ZZ19:=-243.1;
ZZ21:=-460.5;
ZZ25:=-589;
ZZ29:=-722.1;
ZZ30:=-574;
ZZ32:=-492.8;
ZZ33:=-422.3;
ZZ34:=-411.5;
ZZ36:=-333.3;
ZZ38:=-261.2;
ZZ39:=-214;
ZZ41:=-469.1;
ZZ42:=-524.5;
ZZ45:=-579.4;
ZZ46:=-590.2;
ZZ47:=-633.4;
ZZ48:=-686;
ZZ49:=-704.5;
ZZ61:=-320.1;
ZZ67:=-309.8;
ZZ69:=-297.5;




  ENDPROC


ENDMODULE
